        (* Output: *)
        (* judge = *)
        (* 1 *)
        (* 'NearZero:15' judge = norm(near) < 1e-6; *)
        se3mat_0[0] := V[0];
        se3mat_0[1] := V[1];
        se3mat_0[2] := V[2];
        e_theta := norm(x := se3mat_0);
        IF ABS(e_theta) < 1.0E-6 THEN 
            (* 'MatrixExp6:24' T = [eye(3), se3mat(1: 3, 4); 0, 0, 0, 1]; *)
            i0_eye();
            tmp_0 := i0_eye.I;
            FOR Slist_tmp_0 := 0 TO 2 DO 
                R_tmp := DWORD_TO_DINT(SHL(DINT_TO_DWORD(Slist_tmp_0), 2));
                a[R_tmp] := tmp_0[3 * Slist_tmp_0];
                a[R_tmp + 1] := tmp_0[(3 * Slist_tmp_0) + 1];
                a[R_tmp + 2] := tmp_0[(3 * Slist_tmp_0) + 2];
                a[Slist_tmp_0 + 12] := se3mat[Slist_tmp_0 + 12];
            END_FOR;
            a[3] := 0.0;
            a[7] := 0.0;
            a[11] := 0.0;
            a[15] := 1.0;
        ELSE 
            (* 'MatrixExp6:25' else *)
            (* 'MatrixExp6:26' [omghat, theta] = AxisAng3(omgtheta); *)
            (* *** CHAPTER 3: RIGID-BODY MOTIONS *** *)
            (* Takes A 3-vector of exponential coordinates for rotation. *)
            (* Returns the unit rotation axis omghat and the corresponding rotation  *)
            (* angle theta. *)
            (* Example Input: *)
            
            (* clear; clc; *)
            (* expc3 = [1; 2; 3]; *)
            (* [omghat, theta] = AxisAng3(expc3)   *)
            
            (* Output: *)
            (* omghat = *)
            (* 0.2673 *)
            (* 0.5345 *)
            (* 0.8018 *)
            (* theta = *)
            (* 3.7417 *)
            (* 'AxisAng3:20' theta = norm(expc3); *)
            (* 'AxisAng3:21' omghat = expc3 / theta; *)
            (* 'MatrixExp6:27' omgmat = se3mat(1: 3, 1: 3) / theta; *)
            FOR Slist_tmp_0 := 0 TO 2 DO 
                omgmat_tmp := DWORD_TO_DINT(SHL(DINT_TO_DWORD(Slist_tmp_0), 2));
                omgmat[3 * Slist_tmp_0] := se3mat[omgmat_tmp] / e_theta;
                omgmat[(3 * Slist_tmp_0) + 1] := se3mat[omgmat_tmp + 1] / e_theta;
                omgmat[(3 * Slist_tmp_0) + 2] := se3mat[omgmat_tmp + 2] / e_theta;
            END_FOR;
            (* 'MatrixExp6:28' T = [MatrixExp3(se3mat(1: 3, 1: 3)), ... *)
            (* 'MatrixExp6:29'          (eye(3) * theta + (1 - cos(theta)) * omgmat ... *)
            (* 'MatrixExp6:30'           + (theta - sin(theta)) * omgmat * omgmat) ... *)
            (* 'MatrixExp6:31'             * se3mat(1: 3, 4) / theta; *)
            (* 'MatrixExp6:32'          0, 0, 0, 1]; *)
            thetalist0_0 := 1.0 - COS(e_theta);
            g_a := e_theta - SIN(e_theta);
            (* *** CHAPTER 3: RIGID-BODY MOTIONS *** *)
            (* Takes a 3x3 so(3) representation of exponential coordinates. *)
            (* Returns R in SO(3) that is achieved by rotating about omghat by theta  *)
            (* from an initial orientation R = I. *)
            (* Example Input: *)
            
            (* clear; clc; *)
            (* so3mat = [[0, -3, 2]; [3, 0, -1]; [-2, 1, 0]]; *)
            (* R = MatrixExp3(so3mat)   *)
            
            (* Output: *)
            (* R = *)
            (* -0.6949    0.7135    0.0893 *)
            (* -0.1920   -0.3038    0.9332 *)
            (* 0.6930    0.6313    0.3481 *)
            (* 'MatrixExp3:18' omgtheta = so3ToVec(so3mat); *)
            (* *** CHAPTER 3: RIGID-BODY MOTIONS *** *)
            (* Takes a 3x3 skew-symmetric matrix (an element of so(3)). *)
            (* Returns the corresponding 3-vector (angular velocity). *)
            (* Example Input:  *)
            
            (* clear; clc; *)
            (* so3mat = [[0, -3, 2]; [3, 0, -1]; [-2, 1, 0]]; *)
            (* omg = so3ToVec(so3mat)   *)
            
            (* Output: *)
            (* omg = *)
            (* 1 *)
            (* 2 *)
            (* 3 *)
            (* 'so3ToVec:17' omg = [so3mat(3, 2); so3mat(1, 3); so3mat(2, 1)]; *)
            (* 'MatrixExp3:19' if NearZero(norm(omgtheta)) *)
            (* *** BASIC HELPER FUNCTIONS *** *)
            (* Takes a scalar. *)
            (* Checks if the scalar is small enough to be neglected. *)
            (* Example Input: *)
            
            (* clear; clc; *)
            (* near = -1e-7; *)
            (* judge = NearZero(near) *)
            
            (* Output: *)
            (* judge = *)
            (* 1 *)
            (* 'NearZero:15' judge = norm(near) < 1e-6; *)
            se3mat_0[0] := V[0];
            se3mat_0[1] := V[1];
            se3mat_0[2] := V[2];
            h_theta := norm(x := se3mat_0);
            IF ABS(h_theta) < 1.0E-6 THEN 
                (* 'MatrixExp3:20' R = eye(3); *)
                i0_eye();
                b_R := i0_eye.I;
            ELSE 
                (* 'MatrixExp3:21' else *)
                (* 'MatrixExp3:22' [omghat, theta] = AxisAng3(omgtheta); *)
                (* *** CHAPTER 3: RIGID-BODY MOTIONS *** *)
                (* Takes A 3-vector of exponential coordinates for rotation. *)
                (* Returns the unit rotation axis omghat and the corresponding rotation  *)
                (* angle theta. *)
                (* Example Input: *)
                
                (* clear; clc; *)
                (* expc3 = [1; 2; 3]; *)
                (* [omghat, theta] = AxisAng3(expc3)   *)
                
                (* Output: *)
                (* omghat = *)
                (* 0.2673 *)
                (* 0.5345 *)
                (* 0.8018 *)
                (* theta = *)
                (* 3.7417 *)
                (* 'AxisAng3:20' theta = norm(expc3); *)
                (* 'AxisAng3:21' omghat = expc3 / theta; *)
                (* 'MatrixExp3:23' omgmat = so3mat / theta; *)
                FOR Slist_tmp_0 := 0 TO 2 DO 
                    omgmat_tmp := DWORD_TO_DINT(SHL(DINT_TO_DWORD(Slist_tmp_0), 2));
                    b_omgmat[3 * Slist_tmp_0] := se3mat[omgmat_tmp] / h_theta;
                    b_omgmat[(3 * Slist_tmp_0) + 1] := se3mat[omgmat_tmp + 1] / h_theta;
                    b_omgmat[(3 * Slist_tmp_0) + 2] := se3mat[omgmat_tmp + 2] / h_theta;
                END_FOR;
                (* 'MatrixExp3:24' R = eye(3) + sin(theta) * omgmat + (1 - cos(theta)) * omgmat * omgmat; *)
                l_a := SIN(h_theta);
                x_tmp := COS(h_theta);
                i0_eye();
                tmp_0 := i0_eye.I;
                FOR Slist_tmp_0 := 0 TO 2 DO 
                    FOR omgmat_tmp := 0 TO 2 DO 
                        R_tmp := (3 * omgmat_tmp) + Slist_tmp_0;
                        b_R[R_tmp] := (((((1.0 - x_tmp) * b_omgmat[Slist_tmp_0 + 3]) * b_omgmat[(3 * omgmat_tmp) + 1]) + (((1.0 - x_tmp) * b_omgmat[Slist_tmp_0]) * b_omgmat[3 * omgmat_tmp])) + ((b_omgmat[Slist_tmp_0 + 6] * (1.0 - x_tmp)) * b_omgmat[(3 * omgmat_tmp) + 2])) + ((b_omgmat[R_tmp] * l_a) + tmp_0[R_tmp]);
                    END_FOR;
                END_FOR;
            END_IF;
            FOR Slist_tmp_0 := 0 TO 2 DO 
                l_a := 0.0;
                FOR omgmat_tmp := 0 TO 2 DO 
                    R_tmp := (3 * omgmat_tmp) + Slist_tmp_0;
                    l_a := ((((((omgmat[Slist_tmp_0 + 3] * g_a) * omgmat[(3 * omgmat_tmp) + 1]) + ((g_a * omgmat[Slist_tmp_0]) * omgmat[3 * omgmat_tmp])) + ((omgmat[Slist_tmp_0 + 6] * g_a) * omgmat[(3 * omgmat_tmp) + 2])) + ((SINT_TO_LREAL(p_a[R_tmp]) * e_theta) + (omgmat[R_tmp] * thetalist0_0))) * se3mat[omgmat_tmp + 12]) + l_a;
                    a[omgmat_tmp + (Slist_tmp_0 * 4)] := b_R[(3 * Slist_tmp_0) + omgmat_tmp];
                END_FOR;
                a[Slist_tmp_0 + 12] := l_a / e_theta;
            END_FOR;
            a[3] := 0.0;
            a[7] := 0.0;
            a[11] := 0.0;
            a[15] := 1.0;
        END_IF;
        FOR Slist_tmp_0 := 0 TO 3 DO 
            FOR omgmat_tmp := 0 TO 3 DO 
                a_tmp_tmp := DWORD_TO_DINT(SHL(DINT_TO_DWORD(omgmat_tmp), 2));
                R_tmp := Slist_tmp_0 + a_tmp_tmp;
                b_T[R_tmp] := 0.0;
                b_T[R_tmp] := b_T[R_tmp] + (a[a_tmp_tmp] * a_0[Slist_tmp_0]);
                b_T[R_tmp] := (a[a_tmp_tmp + 1] * a_0[Slist_tmp_0 + 4]) + b_T[R_tmp];
                b_T[R_tmp] := (a[a_tmp_tmp + 2] * a_0[Slist_tmp_0 + 8]) + b_T[R_tmp];
                b_T[R_tmp] := (a[a_tmp_tmp + 3] * a_0[Slist_tmp_0 + 12]) + b_T[R_tmp];
            END_FOR;
        END_FOR;
        FOR Slist_tmp_0 := 0 TO 15 DO 
            a_0[Slist_tmp_0] := b_T[Slist_tmp_0];
        END_FOR;
        (* 'JacobianSpace:31' Js(:, i) = Adjoint(T) * Slist(:, i); *)
        (* *** CHAPTER 3: RIGID-BODY MOTIONS *** *)
        (* Takes T a transformation matrix SE3.  *)
        (* Returns the corresponding 6x6 adjoint representation [AdT]. *)
        (* Example Input: *)
        
        (* clear; clc; *)
        (* T = [[1, 0, 0, 0]; [0, 0, -1, 0]; [0, 1, 0, 3]; [0, 0, 0, 1]]; *)
        (* AdT = Adjoint(T) *)
        
        (* Output: *)
        (* AdT = *)
        (* 1     0     0     0     0     0 *)
        (* 0     0    -1     0     0     0 *)
        (* 0     1     0     0     0     0 *)
        (* 0     0     3     1     0     0 *)
        (* 3     0     0     0     0    -1 *)
        (* 0     0     0     0     1     0 *)
        (* 'Adjoint:20' [R, p] = TransToRp(T); *)
        (* *** CHAPTER 3: RIGID-BODY MOTIONS *** *)
        (* Takes the transformation matrix T in SE(3)  *)
        (* Returns R: the corresponding rotation matrix *)
        (* p: the corresponding position vector . *)
        (* Example Input: *)
        
        (* clear; clc; *)
        (* T = [[1, 0, 0, 0]; [0, 0, -1, 0]; [0, 1, 0, 3]; [0, 0, 0, 1]]; *)
        (* [R, p] = TransToRp(T) *)
        
        (* Output: *)
        (* R = *)
        (* 1     0     0 *)
        (* 0     0    -1 *)
        (* 0     1     0 *)
        (* p = *)
        (* 0 *)
        (* 0 *)
        (* 3 *)
        (* 'TransToRp:22' R = T(1: 3, 1: 3); *)
        (* 'TransToRp:23' p = T(1: 3, 4); *)
        (* 'Adjoint:21' AdT = [R, zeros(3); VecToso3(p) * R, R]; *)
        (* *** CHAPTER 3: RIGID-BODY MOTIONS *** *)
        (* Takes a 3-vector (angular velocity). *)
        (* Returns the skew symmetric matrix in so(3). *)
        (* Example Input: *)
        
        (* clear; clc; *)
        (* omg = [1; 2; 3]; *)
        (* so3mat = VecToso3(omg) *)
        
        (* Output: *)
        (* so3mat = *)
        (* 0    -3     2 *)
        (* 3     0    -1 *)
        (* -2     1     0 *)
        (* 'VecToso3:17' so3mat = [0, -omg(3), omg(2); omg(3), 0, -omg(1); -omg(2), omg(1), 0]; *)
        tmp_3[3] :=  -a_0[14];
        tmp_3[6] := a_0[13];
        tmp_3[1] := a_0[14];
        tmp_3[7] :=  -a_0[12];
        tmp_3[2] :=  -a_0[13];
        tmp_3[5] := a_0[12];
        FOR Slist_tmp_0 := 0 TO 2 DO 
            FOR omgmat_tmp := 0 TO 2 DO 
                R_tmp := Slist_tmp_0 + (3 * omgmat_tmp);
                tmp_0[R_tmp] := 0.0;
                a_tmp_tmp := DWORD_TO_DINT(SHL(DINT_TO_DWORD(omgmat_tmp), 2));
                tmp_0[R_tmp] := tmp_0[R_tmp] + (a_0[a_tmp_tmp] * tmp_3[Slist_tmp_0]);
                tmp_0[R_tmp] := (a_0[a_tmp_tmp + 1] * tmp_3[Slist_tmp_0 + 3]) + tmp_0[R_tmp];
                tmp_0[R_tmp] := (a_0[a_tmp_tmp + 2] * tmp_3[Slist_tmp_0 + 6]) + tmp_0[R_tmp];
                Tsb_0[omgmat_tmp + (6 * Slist_tmp_0)] := a_0[(Slist_tmp_0 * 4) + omgmat_tmp];
                Tsb_0[omgmat_tmp + (6 * (Slist_tmp_0 + 3))] := 0.0;
            END_FOR;
        END_FOR;
        FOR Slist_tmp_0 := 0 TO 2 DO 
            Tsb_0[(6 * Slist_tmp_0) + 3] := tmp_0[3 * Slist_tmp_0];
            R_tmp := DWORD_TO_DINT(SHL(DINT_TO_DWORD(Slist_tmp_0), 2));
            omgmat_tmp := 6 * (Slist_tmp_0 + 3);
            Tsb_0[omgmat_tmp + 3] := a_0[R_tmp];
            Tsb_0[(6 * Slist_tmp_0) + 4] := tmp_0[(3 * Slist_tmp_0) + 1];
            Tsb_0[omgmat_tmp + 4] := a_0[R_tmp + 1];
            Tsb_0[(6 * Slist_tmp_0) + 5] := tmp_0[(3 * Slist_tmp_0) + 2];
            Tsb_0[omgmat_tmp + 5] := a_0[R_tmp + 2];
        END_FOR;
        FOR Slist_tmp_0 := 0 TO 5 DO 
            R_tmp := 6 * (d_i + 1);
            a_tmp_tmp := Slist_tmp_0 + R_tmp;
            Js[a_tmp_tmp] := 0.0;
            FOR omgmat_tmp := 0 TO 5 DO 
                Js[a_tmp_tmp] := (Slist[R_tmp + omgmat_tmp] * Tsb_0[(6 * omgmat_tmp) + Slist_tmp_0]) + Js[a_tmp_tmp];
            END_FOR;
        END_FOR;
    END_FOR;
    i0_pinv(A := Js);
    tmp_1 := i0_pinv.X;
    FOR Slist_tmp_0 := 0 TO 4 DO 
        l_a := 0.0;
        FOR omgmat_tmp := 0 TO 5 DO 
            l_a := (tmp_1[(5 * omgmat_tmp) + Slist_tmp_0] * Vs[omgmat_tmp]) + l_a;
        END_FOR;
        thetalist0[Slist_tmp_0] := thetalist0[Slist_tmp_0] + l_a;
    END_FOR;
    (* 'IKinSpace:57' thetalistDot = pinv(JacobianSpace(Slist, thetalist)) * Vs; *)
    (* *** CHAPTER 5: VELOCITY KINEMATICS AND STATICS *** *)
    (* Takes Slist: The joint screw axes in the space frame when the manipulator *)
    (* is at the home position, in the format of a matrix with the *)
    (* screw axes as the columns, *)
    (* thetalist: A list of joint coordinates.  *)
    (* Returns the corresponding space Jacobian (6xn real numbers). *)
    (* Example Input: *)
    
    (* clear; clc; *)
    (* Slist = [[0; 0; 1;   0; 0.2; 0.2], ... *)
    (* [1; 0; 0;   2;   0;   3], ... *)
    (* [0; 1; 0;   0;   2;   1], ... *)
    (* [1; 0; 0; 0.2; 0.3; 0.4]]; *)
    (* thetalist = [0.2; 1.1; 0.1; 1.2]; *)
    (* Js = JacobianSpace(Slist, thetalist) *)
    
    (* Output: *)
    (* Js = *)
    (* 0    0.9801   -0.0901    0.9575 *)
    (* 0    0.1987    0.4446    0.2849 *)
    (* 1.0000         0    0.8912   -0.0453 *)
    (* 0    1.9522   -2.2164   -0.5116 *)
    (* 0.2000    0.4365   -2.4371    2.7754 *)
    (* 0.2000    2.9603    3.2357    2.2251 *)
    (* 'JacobianSpace:27' Js = Slist; *)
    (* 'JacobianSpace:28' T = eye(4); *)
    (* 'JacobianSpace:29' for i = 2: length(thetalist) *)
    (* 'IKinSpace:58' i = i + 1; *)
    i := i + 1;
    (* 'IKinSpace:59' Tsb = FKinSpace(M, Slist, thetalist); *)
    FOR Slist_tmp_0 := 0 TO 15 DO 
        Tsb[Slist_tmp_0] := M[Slist_tmp_0];
    END_FOR;
    (* *** CHAPTER 4: FORWARD KINEMATICS *** *)
    (* Takes M: the home configuration (position and orientation) of the  *)
    (* end-effector, *)
    (* Slist: The joint screw axes in the space frame when the manipulator *)
    (* is at the home position, *)
    (* thetalist: A list of joint coordinates. *)
    (* Returns T in SE(3) representing the end-effector frame, when the joints  *)
    (* are at the specified coordinates (i.t.o Space Frame). *)
    (* Example Inputs: *)
    
    (* clear; clc; *)
    (* M = [[-1, 0, 0, 0]; [0, 1, 0, 6]; [0, 0, -1, 2]; [0, 0, 0, 1]]; *)
    (* Slist = [[0; 0;  1;  4; 0;    0], ... *)
    (* [0; 0;  0;  0; 1;    0], ... *)
    (* [0; 0; -1; -6; 0; -0.1]]; *)
    (* thetalist =[pi / 2; 3; pi]; *)
    (* T = FKinSpace(M, Slist, thetalist) *)
    
    (* Output: *)
    (* T = *)
    (* -0.0000    1.0000         0   -5.0000 *)
    (* 1.0000    0.0000         0    4.0000 *)
    (* 0         0   -1.0000    1.6858 *)
    (* 0         0         0    1.0000 *)
    (* 'FKinSpace:27' T = M; *)
    (* 'FKinSpace:28' for i = size(thetalist,1): -1: 1 *)
    se3mat[0] := 0.0;
    se3mat[5] := 0.0;
    se3mat[10] := 0.0;
    se3mat[3] := 0.0;
    se3mat[7] := 0.0;
    se3mat[11] := 0.0;
    se3mat[15] := 0.0;
    FOR e_i := 0 TO 4 DO 
        (* 'FKinSpace:29' T = MatrixExp6(VecTose3(Slist(:, i) * thetalist(i))) * T; *)
        thetalist0_0 := thetalist0[4 - e_i];
        FOR Slist_tmp_0 := 0 TO 5 DO 
            V[Slist_tmp_0] := Slist[((4 - e_i) * 6) + Slist_tmp_0] * thetalist0_0;
        END_FOR;
        (* *** CHAPTER 3: RIGID-BODY MOTIONS *** *)
        (* Takes a 6-vector (representing a spatial velocity). *)
        (* Returns the corresponding 4x4 se(3) matrix. *)
        (* Example Input: *)
        
        (* clear; clc; *)
        (* V = [1; 2; 3; 4; 5; 6]; *)
        (* se3mat = VecTose3(V) *)
        
        (* Output: *)
        (* se3mat = *)
        (* 0    -3     2     4 *)
        (* 3     0    -1     5 *)
        (* -2     1     0     6 *)
        (* 0     0     0     0  *)
        (* 'VecTose3:18' se3mat = [VecToso3(V(1: 3)), V(4: 6); 0, 0, 0, 0]; *)
        (* *** CHAPTER 3: RIGID-BODY MOTIONS *** *)
        (* Takes a 3-vector (angular velocity). *)
        (* Returns the skew symmetric matrix in so(3). *)
        (* Example Input: *)
        
        (* clear; clc; *)
        (* omg = [1; 2; 3]; *)
        (* so3mat = VecToso3(omg) *)
        
        (* Output: *)
        (* so3mat = *)
        (* 0    -3     2 *)
        (* 3     0    -1 *)
        (* -2     1     0 *)
        (* 'VecToso3:17' so3mat = [0, -omg(3), omg(2); omg(3), 0, -omg(1); -omg(2), omg(1), 0]; *)
        se3mat[4] :=  -V[2];
        se3mat[8] := V[1];
        se3mat[1] := V[2];
        se3mat[9] :=  -V[0];
        se3mat[2] :=  -V[1];
        se3mat[6] := V[0];
        se3mat[12] := V[3];
        se3mat[13] := V[4];
        se3mat[14] := V[5];
        (* *** CHAPTER 3: RIGID-BODY MOTIONS *** *)
        (* Takes a se(3) representation of exponential coordinates. *)
        (* Returns a T matrix in SE(3) that is achieved by traveling along/about the  *)
        (* screw axis S for a distance theta from an initial configuration T = I. *)
        (* Example Input: *)
        
        (* clear; clc; *)
        (* se3mat = [ 0,      0,       0,      0; *)
        (* 0,      0, -1.5708, 2.3562; *)
        (* 0, 1.5708,       0, 2.3562; *)
        (* 0,      0,       0,      0] *)
        (* T = MatrixExp6(se3mat) *)
        
        (* Output: *)
        (* T = *)
        (* 1.0000         0         0         0 *)
        (* 0    0.0000   -1.0000   -0.0000 *)
        (* 0    1.0000    0.0000    3.0000 *)
        (* 0         0         0    1.0000  *)
        (* 'MatrixExp6:22' omgtheta = so3ToVec(se3mat(1: 3, 1: 3)); *)
        (* *** CHAPTER 3: RIGID-BODY MOTIONS *** *)
        (* Takes a 3x3 skew-symmetric matrix (an element of so(3)). *)
        (* Returns the corresponding 3-vector (angular velocity). *)
        (* Example Input:  *)
        
        (* clear; clc; *)
        (* so3mat = [[0, -3, 2]; [3, 0, -1]; [-2, 1, 0]]; *)
        (* omg = so3ToVec(so3mat)   *)
        
        (* Output: *)
        (* omg = *)
        (* 1 *)
        (* 2 *)
        (* 3 *)
        (* 'so3ToVec:17' omg = [so3mat(3, 2); so3mat(1, 3); so3mat(2, 1)]; *)
        omgtheta[0] := V[0];
        omgtheta[1] := V[1];
        omgtheta[2] := V[2];
        (* 'MatrixExp6:23' if NearZero(norm(omgtheta)) *)
        (* *** BASIC HELPER FUNCTIONS *** *)
        (* Takes a scalar. *)
        (* Checks if the scalar is small enough to be neglected. *)
        (* Example Input: *)
        
        (* clear; clc; *)
        (* near = -1e-7; *)
        (* judge = NearZero(near) *)
        
        (* Output: *)
        (* judge = *)
        (* 1 *)
        (* 'NearZero:15' judge = norm(near) < 1e-6; *)
        f_theta := norm(x := omgtheta);
        IF ABS(f_theta) < 1.0E-6 THEN 
            (* 'MatrixExp6:24' T = [eye(3), se3mat(1: 3, 4); 0, 0, 0, 1]; *)
            i0_eye();
            tmp_0 := i0_eye.I;
            FOR Slist_tmp_0 := 0 TO 2 DO 
                R_tmp := DWORD_TO_DINT(SHL(DINT_TO_DWORD(Slist_tmp_0), 2));
                a[R_tmp] := tmp_0[3 * Slist_tmp_0];
                a[R_tmp + 1] := tmp_0[(3 * Slist_tmp_0) + 1];
                a[R_tmp + 2] := tmp_0[(3 * Slist_tmp_0) + 2];
                a[Slist_tmp_0 + 12] := se3mat[Slist_tmp_0 + 12];
            END_FOR;
            a[3] := 0.0;
            a[7] := 0.0;
            a[11] := 0.0;
            a[15] := 1.0;
        ELSE 
            (* 'MatrixExp6:25' else *)
            (* 'MatrixExp6:26' [omghat, theta] = AxisAng3(omgtheta); *)
            (* *** CHAPTER 3: RIGID-BODY MOTIONS *** *)
            (* Takes A 3-vector of exponential coordinates for rotation. *)
            (* Returns the unit rotation axis omghat and the corresponding rotation  *)
            (* angle theta. *)
            (* Example Input: *)
            
            (* clear; clc; *)
            (* expc3 = [1; 2; 3]; *)
            (* [omghat, theta] = AxisAng3(expc3)   *)
            
            (* Output: *)
            (* omghat = *)
            (* 0.2673 *)
            (* 0.5345 *)
            (* 0.8018 *)
            (* theta = *)
            (* 3.7417 *)
            (* 'AxisAng3:20' theta = norm(expc3); *)
            (* 'AxisAng3:21' omghat = expc3 / theta; *)
            (* 'MatrixExp6:27' omgmat = se3mat(1: 3, 1: 3) / theta; *)
            FOR Slist_tmp_0 := 0 TO 2 DO 
                omgmat_tmp := DWORD_TO_DINT(SHL(DINT_TO_DWORD(Slist_tmp_0), 2));
                omgmat[3 * Slist_tmp_0] := se3mat[omgmat_tmp] / f_theta;
                omgmat[(3 * Slist_tmp_0) + 1] := se3mat[omgmat_tmp + 1] / f_theta;
                omgmat[(3 * Slist_tmp_0) + 2] := se3mat[omgmat_tmp + 2] / f_theta;
            END_FOR;
            (* 'MatrixExp6:28' T = [MatrixExp3(se3mat(1: 3, 1: 3)), ... *)
            (* 'MatrixExp6:29'          (eye(3) * theta + (1 - cos(theta)) * omgmat ... *)
            (* 'MatrixExp6:30'           + (theta - sin(theta)) * omgmat * omgmat) ... *)
            (* 'MatrixExp6:31'             * se3mat(1: 3, 4) / theta; *)
            (* 'MatrixExp6:32'          0, 0, 0, 1]; *)
            thetalist0_0 := 1.0 - COS(f_theta);
            g_a := f_theta - SIN(f_theta);
            (* *** CHAPTER 3: RIGID-BODY MOTIONS *** *)
            (* Takes a 3x3 so(3) representation of exponential coordinates. *)
            (* Returns R in SO(3) that is achieved by rotating about omghat by theta  *)
            (* from an initial orientation R = I. *)
            (* Example Input: *)
            
            (* clear; clc; *)
            (* so3mat = [[0, -3, 2]; [3, 0, -1]; [-2, 1, 0]]; *)
            (* R = MatrixExp3(so3mat)   *)
            
            (* Output: *)
            (* R = *)
            (* -0.6949    0.7135    0.0893 *)
            (* -0.1920   -0.3038    0.9332 *)
            (* 0.6930    0.6313    0.3481 *)
            (* 'MatrixExp3:18' omgtheta = so3ToVec(so3mat); *)
            (* *** CHAPTER 3: RIGID-BODY MOTIONS *** *)
            (* Takes a 3x3 skew-symmetric matrix (an element of so(3)). *)
            (* Returns the corresponding 3-vector (angular velocity). *)
            (* Example Input:  *)
            
            (* clear; clc; *)
            (* so3mat = [[0, -3, 2]; [3, 0, -1]; [-2, 1, 0]]; *)
            (* omg = so3ToVec(so3mat)   *)
            
            (* Output: *)
            (* omg = *)
            (* 1 *)
            (* 2 *)
            (* 3 *)
            (* 'so3ToVec:17' omg = [so3mat(3, 2); so3mat(1, 3); so3mat(2, 1)]; *)
            (* 'MatrixExp3:19' if NearZero(norm(omgtheta)) *)
            (* *** BASIC HELPER FUNCTIONS *** *)
            (* Takes a scalar. *)
            (* Checks if the scalar is small enough to be neglected. *)
            (* Example Input: *)
            
            (* clear; clc; *)
            (* near = -1e-7; *)
            (* judge = NearZero(near) *)
            
            (* Output: *)
            (* judge = *)
            (* 1 *)
            (* 'NearZero:15' judge = norm(near) < 1e-6; *)
            se3mat_0[0] := V[0];
            se3mat_0[1] := V[1];
            se3mat_0[2] := V[2];
            j_theta := norm(x := se3mat_0);
            IF ABS(j_theta) < 1.0E-6 THEN 
                (* 'MatrixExp3:20' R = eye(3); *)
                i0_eye();
                b_R := i0_eye.I;
            ELSE 
                (* 'MatrixExp3:21' else *)
                (* 'MatrixExp3:22' [omghat, theta] = AxisAng3(omgtheta); *)
                (* *** CHAPTER 3: RIGID-BODY MOTIONS *** *)
                (* Takes A 3-vector of exponential coordinates for rotation. *)
                (* Returns the unit rotation axis omghat and the corresponding rotation  *)
                (* angle theta. *)
                (* Example Input: *)
                
                (* clear; clc; *)
                (* expc3 = [1; 2; 3]; *)
                (* [omghat, theta] = AxisAng3(expc3)   *)
                
                (* Output: *)
                (* omghat = *)
                (* 0.2673 *)
                (* 0.5345 *)
                (* 0.8018 *)
                (* theta = *)
                (* 3.7417 *)
                (* 'AxisAng3:20' theta = norm(expc3); *)
                (* 'AxisAng3:21' omghat = expc3 / theta; *)
                (* 'MatrixExp3:23' omgmat = so3mat / theta; *)
                FOR Slist_tmp_0 := 0 TO 2 DO 
                    omgmat_tmp := DWORD_TO_DINT(SHL(DINT_TO_DWORD(Slist_tmp_0), 2));
                    b_omgmat[3 * Slist_tmp_0] := se3mat[omgmat_tmp] / j_theta;
                    b_omgmat[(3 * Slist_tmp_0) + 1] := se3mat[omgmat_tmp + 1] / j_theta;
                    b_omgmat[(3 * Slist_tmp_0) + 2] := se3mat[omgmat_tmp + 2] / j_theta;
                END_FOR;
                (* 'MatrixExp3:24' R = eye(3) + sin(theta) * omgmat + (1 - cos(theta)) * omgmat * omgmat; *)
                l_a := SIN(j_theta);
                x_tmp := COS(j_theta);
                i0_eye();
                tmp_0 := i0_eye.I;
                FOR Slist_tmp_0 := 0 TO 2 DO 
                    FOR omgmat_tmp := 0 TO 2 DO 
                        R_tmp := (3 * omgmat_tmp) + Slist_tmp_0;
                        b_R[R_tmp] := (((((1.0 - x_tmp) * b_omgmat[Slist_tmp_0 + 3]) * b_omgmat[(3 * omgmat_tmp) + 1]) + (((1.0 - x_tmp) * b_omgmat[Slist_tmp_0]) * b_omgmat[3 * omgmat_tmp])) + ((b_omgmat[Slist_tmp_0 + 6] * (1.0 - x_tmp)) * b_omgmat[(3 * omgmat_tmp) + 2])) + ((b_omgmat[R_tmp] * l_a) + tmp_0[R_tmp]);
                    END_FOR;
                END_FOR;
            END_IF;
            FOR Slist_tmp_0 := 0 TO 2 DO 
                l_a := 0.0;
                FOR omgmat_tmp := 0 TO 2 DO 
                    R_tmp := (3 * omgmat_tmp) + Slist_tmp_0;
                    l_a := ((((((omgmat[Slist_tmp_0 + 3] * g_a) * omgmat[(3 * omgmat_tmp) + 1]) + ((g_a * omgmat[Slist_tmp_0]) * omgmat[3 * omgmat_tmp])) + ((omgmat[Slist_tmp_0 + 6] * g_a) * omgmat[(3 * omgmat_tmp) + 2])) + ((SINT_TO_LREAL(p_a[R_tmp]) * f_theta) + (omgmat[R_tmp] * thetalist0_0))) * se3mat[omgmat_tmp + 12]) + l_a;
                    a[omgmat_tmp + (Slist_tmp_0 * 4)] := b_R[(3 * Slist_tmp_0) + omgmat_tmp];
                END_FOR;
                a[Slist_tmp_0 + 12] := l_a / f_theta;
            END_FOR;
            a[3] := 0.0;
            a[7] := 0.0;
            a[11] := 0.0;
            a[15] := 1.0;
        END_IF;
        FOR Slist_tmp_0 := 0 TO 3 DO 
            FOR omgmat_tmp := 0 TO 3 DO 
                a_tmp_tmp := DWORD_TO_DINT(SHL(DINT_TO_DWORD(omgmat_tmp), 2));
                R_tmp := Slist_tmp_0 + a_tmp_tmp;
                a_0[R_tmp] := 0.0;
                a_0[R_tmp] := a_0[R_tmp] + (Tsb[a_tmp_tmp] * a[Slist_tmp_0]);
                a_0[R_tmp] := (Tsb[a_tmp_tmp + 1] * a[Slist_tmp_0 + 4]) + a_0[R_tmp];
                a_0[R_tmp] := (Tsb[a_tmp_tmp + 2] * a[Slist_tmp_0 + 8]) + a_0[R_tmp];
                a_0[R_tmp] := (Tsb[a_tmp_tmp + 3] * a[Slist_tmp_0 + 12]) + a_0[R_tmp];
            END_FOR;
        END_FOR;
        FOR Slist_tmp_0 := 0 TO 15 DO 
            Tsb[Slist_tmp_0] := a_0[Slist_tmp_0];
        END_FOR;
    END_FOR;
    (* 'IKinSpace:60' Vs = Adjoint(Tsb) * se3ToVec(MatrixLog6(TransInv(Tsb) * T)); *)
    (* *** CHAPTER 3: RIGID-BODY MOTIONS *** *)
    (* Takes a transformation matrix T. *)
    (* Returns its inverse.  *)
    (* Uses the structure of transformation matrices to avoid taking a matrix *)
    (* inverse, for efficiency. *)
    (* Example Input: *)
    
    (* clear; clc; *)
    (* T = [[1, 0, 0, 0]; [0, 0, -1, 0]; [0, 1, 0, 3]; [0, 0, 0, 1]]; *)
    (* invT = TransInv(T) *)
    
    (* Ouput: *)
    (* invT = *)
    (* 1     0     0     0 *)
    (* 0     0     1    -3 *)
    (* 0    -1     0     0 *)
    (* 0     0     0     1 *)
    (* 'TransInv:20' [R, p] = TransToRp(T); *)
    (* *** CHAPTER 3: RIGID-BODY MOTIONS *** *)
    (* Takes the transformation matrix T in SE(3)  *)
    (* Returns R: the corresponding rotation matrix *)
    (* p: the corresponding position vector . *)
    (* Example Input: *)
    
    (* clear; clc; *)
    (* T = [[1, 0, 0, 0]; [0, 0, -1, 0]; [0, 1, 0, 3]; [0, 0, 0, 1]]; *)
    (* [R, p] = TransToRp(T) *)
    
    (* Output: *)
    (* R = *)
    (* 1     0     0 *)
    (* 0     0    -1 *)
    (* 0     1     0 *)
    (* p = *)
    (* 0 *)
    (* 0 *)
    (* 3 *)
    (* 'TransToRp:22' R = T(1: 3, 1: 3); *)
    (* 'TransToRp:23' p = T(1: 3, 4); *)
    (* 'TransInv:21' invT = [transpose(R), -transpose(R) * p; 0, 0, 0, 1]; *)
    FOR Slist_tmp_0 := 0 TO 2 DO 
        omgmat[3 * Slist_tmp_0] := Tsb[Slist_tmp_0];
        omgmat[(3 * Slist_tmp_0) + 1] := Tsb[Slist_tmp_0 + 4];
        omgmat[(3 * Slist_tmp_0) + 2] := Tsb[Slist_tmp_0 + 8];
    END_FOR;
    FOR Slist_tmp_0 := 0 TO 8 DO 
        b_R[Slist_tmp_0] :=  -omgmat[Slist_tmp_0];
    END_FOR;
    FOR Slist_tmp_0 := 0 TO 2 DO 
        omgmat_tmp := DWORD_TO_DINT(SHL(DINT_TO_DWORD(Slist_tmp_0), 2));
        se3mat[omgmat_tmp] := omgmat[3 * Slist_tmp_0];
        se3mat[omgmat_tmp + 1] := omgmat[(3 * Slist_tmp_0) + 1];
        se3mat[omgmat_tmp + 2] := omgmat[(3 * Slist_tmp_0) + 2];
        se3mat[Slist_tmp_0 + 12] := (b_R[Slist_tmp_0 + 6] * Tsb[14]) + ((b_R[Slist_tmp_0 + 3] * Tsb[13]) + (b_R[Slist_tmp_0] * Tsb[12]));
    END_FOR;
    se3mat[3] := 0.0;
    se3mat[7] := 0.0;
    se3mat[11] := 0.0;
    se3mat[15] := 1.0;
    FOR Slist_tmp_0 := 0 TO 3 DO 
        FOR omgmat_tmp := 0 TO 3 DO 
            a_tmp_tmp := DWORD_TO_DINT(SHL(DINT_TO_DWORD(omgmat_tmp), 2));
            R_tmp := Slist_tmp_0 + a_tmp_tmp;
            a_0[R_tmp] := 0.0;
            a_0[R_tmp] := a_0[R_tmp] + (T[a_tmp_tmp] * se3mat[Slist_tmp_0]);
            a_0[R_tmp] := (T[a_tmp_tmp + 1] * se3mat[Slist_tmp_0 + 4]) + a_0[R_tmp];
            a_0[R_tmp] := (T[a_tmp_tmp + 2] * se3mat[Slist_tmp_0 + 8]) + a_0[R_tmp];
            a_0[R_tmp] := (T[a_tmp_tmp + 3] * se3mat[Slist_tmp_0 + 12]) + a_0[R_tmp];
        END_FOR;
    END_FOR;
    (* *** CHAPTER 3: RIGID-BODY MOTIONS *** *)
    (* Takes a transformation matrix T in SE(3). *)
    (* Returns the corresponding se(3) representation of exponential  *)
    (* coordinates. *)
    (* Example Input: *)
    
    (* clear; clc; *)
    (* T = [[1, 0, 0, 0]; [0, 0, -1, 0]; [0, 1, 0, 3]; [0, 0, 0, 1]]; *)
    (* expmat = MatrixLog6(T) *)
    
    (* Output: *)
    (* expc6 = *)
    (* 0         0         0         0 *)
    (* 0         0   -1.5708    2.3562 *)
    (* 0    1.5708         0    2.3562 *)
    (* 0         0         0         0 *)
    (* 'MatrixLog6:19' [R, p] = TransToRp(T); *)
    (* *** CHAPTER 3: RIGID-BODY MOTIONS *** *)
    (* Takes the transformation matrix T in SE(3)  *)
    (* Returns R: the corresponding rotation matrix *)
    (* p: the corresponding position vector . *)
    (* Example Input: *)
    
    (* clear; clc; *)
    (* T = [[1, 0, 0, 0]; [0, 0, -1, 0]; [0, 1, 0, 3]; [0, 0, 0, 1]]; *)
    (* [R, p] = TransToRp(T) *)
    
    (* Output: *)
    (* R = *)
    (* 1     0     0 *)
    (* 0     0    -1 *)
    (* 0     1     0 *)
    (* p = *)
    (* 0 *)
    (* 0 *)
    (* 3 *)
    (* 'TransToRp:22' R = T(1: 3, 1: 3); *)
    (* 'TransToRp:23' p = T(1: 3, 4); *)
    (* 'MatrixLog6:20' omgmat = MatrixLog3(R); *)
    FOR Slist_tmp_0 := 0 TO 2 DO 
        R_tmp := DWORD_TO_DINT(SHL(DINT_TO_DWORD(Slist_tmp_0), 2));
        b_R[3 * Slist_tmp_0] := a_0[R_tmp];
        b_R[(3 * Slist_tmp_0) + 1] := a_0[R_tmp + 1];
        b_R[(3 * Slist_tmp_0) + 2] := a_0[R_tmp + 2];
    END_FOR;
    i0_MatrixLog3(b_R := b_R);
    omgmat := i0_MatrixLog3.so3mat;
    (* 'MatrixLog6:21' if isequal(omgmat, zeros(3)) *)
    IF isequal(varargin_1 := omgmat, varargin_2 := tmp_4) THEN 
        (* 'MatrixLog6:22' expmat = [zeros(3), T(1: 3, 4); 0, 0, 0, 0]; *)
        FOR Slist_tmp_0 := 0 TO 2 DO 
            omgmat_tmp := DWORD_TO_DINT(SHL(DINT_TO_DWORD(Slist_tmp_0), 2));
            se3mat[omgmat_tmp] := 0.0;
            se3mat[omgmat_tmp + 1] := 0.0;
            se3mat[omgmat_tmp + 2] := 0.0;
            se3mat[Slist_tmp_0 + 12] := a_0[Slist_tmp_0 + 12];
        END_FOR;
        se3mat[3] := 0.0;
        se3mat[7] := 0.0;
        se3mat[11] := 0.0;
        se3mat[15] := 0.0;
    ELSE 
        (* 'MatrixLog6:23' else *)
        (* 'MatrixLog6:24' theta = acos((trace(R) - 1) / 2); *)
        b_theta := ACOS((((a_0[0] + a_0[5]) + a_0[10]) - 1.0) / 2.0);
        (* 'MatrixLog6:25' expmat = [omgmat, (eye(3) - omgmat / 2 ... *)
        (* 'MatrixLog6:26'                       + (1 / theta - cot(theta / 2) / 2) ... *)
        (* 'MatrixLog6:27'                         * omgmat * omgmat / theta) * p; *)
        (* 'MatrixLog6:28'               0, 0, 0, 0]; *)
        thetalist0_0 := (1.0 / b_theta) - ((1.0 / TAN(b_theta / 2.0)) / 2.0);
        i0_eye();
        tmp_0 := i0_eye.I;
        FOR Slist_tmp_0 := 0 TO 2 DO 
            se3mat_0[Slist_tmp_0] := 0.0;
            FOR omgmat_tmp := 0 TO 2 DO 
                se3mat[omgmat_tmp + (Slist_tmp_0 * 4)] := omgmat[(3 * Slist_tmp_0) + omgmat_tmp];
                R_tmp := (3 * omgmat_tmp) + Slist_tmp_0;
                se3mat_0[Slist_tmp_0] := (((((((omgmat[Slist_tmp_0 + 3] * thetalist0_0) * omgmat[(3 * omgmat_tmp) + 1]) + ((thetalist0_0 * omgmat[Slist_tmp_0]) * omgmat[3 * omgmat_tmp])) + ((omgmat[Slist_tmp_0 + 6] * thetalist0_0) * omgmat[(3 * omgmat_tmp) + 2])) / b_theta) + (tmp_0[R_tmp] - (omgmat[R_tmp] / 2.0))) * a_0[omgmat_tmp + 12]) + se3mat_0[Slist_tmp_0];
            END_FOR;
            se3mat[Slist_tmp_0 + 12] := se3mat_0[Slist_tmp_0];
        END_FOR;
        se3mat[3] := 0.0;
        se3mat[7] := 0.0;
        se3mat[11] := 0.0;
        se3mat[15] := 0.0;
    END_IF;
    (* *** CHAPTER 3: RIGID-BODY MOTIONS *** *)
    (* Takes T a transformation matrix SE3.  *)
    (* Returns the corresponding 6x6 adjoint representation [AdT]. *)
    (* Example Input: *)
    
    (* clear; clc; *)
    (* T = [[1, 0, 0, 0]; [0, 0, -1, 0]; [0, 1, 0, 3]; [0, 0, 0, 1]]; *)
    (* AdT = Adjoint(T) *)
    
    (* Output: *)
    (* AdT = *)
    (* 1     0     0     0     0     0 *)
    (* 0     0    -1     0     0     0 *)
    (* 0     1     0     0     0     0 *)
    (* 0     0     3     1     0     0 *)
    (* 3     0     0     0     0    -1 *)
    (* 0     0     0     0     1     0 *)
    (* 'Adjoint:20' [R, p] = TransToRp(T); *)
    (* *** CHAPTER 3: RIGID-BODY MOTIONS *** *)
    (* Takes the transformation matrix T in SE(3)  *)
    (* Returns R: the corresponding rotation matrix *)
    (* p: the corresponding position vector . *)
    (* Example Input: *)
    
    (* clear; clc; *)
    (* T = [[1, 0, 0, 0]; [0, 0, -1, 0]; [0, 1, 0, 3]; [0, 0, 0, 1]]; *)
    (* [R, p] = TransToRp(T) *)
    
    (* Output: *)
    (* R = *)
    (* 1     0     0 *)
    (* 0     0    -1 *)
    (* 0     1     0 *)
    (* p = *)
    (* 0 *)
    (* 0 *)
    (* 3 *)
    (* 'TransToRp:22' R = T(1: 3, 1: 3); *)
    (* 'TransToRp:23' p = T(1: 3, 4); *)
    (* 'Adjoint:21' AdT = [R, zeros(3); VecToso3(p) * R, R]; *)
    (* *** CHAPTER 3: RIGID-BODY MOTIONS *** *)
    (* Takes a 3-vector (angular velocity). *)
    (* Returns the skew symmetric matrix in so(3). *)
    (* Example Input: *)
    
    (* clear; clc; *)
    (* omg = [1; 2; 3]; *)
    (* so3mat = VecToso3(omg) *)
    
    (* Output: *)
    (* so3mat = *)
    (* 0    -3     2 *)
    (* 3     0    -1 *)
    (* -2     1     0 *)
    (* 'VecToso3:17' so3mat = [0, -omg(3), omg(2); omg(3), 0, -omg(1); -omg(2), omg(1), 0]; *)
    (* *** CHAPTER 3: RIGID-BODY MOTIONS *** *)
    (* Takes se3mat a 4x4 se(3) matrix *)
    (* Returns the corresponding 6-vector (representing spatial velocity). *)
    (* Example Input: *)
    
    (* clear; clc; *)
    (* se3mat = [[0, -3, 2, 4]; [3, 0, -1, 5]; [-2, 1, 0, 6]; [0, 0, 0, 0]]; *)
    (* V = se3ToVec(se3mat) *)
    
    (* Output: *)
    (* V = *)
    (* 1 *)
    (* 2 *)
    (* 3 *)
    (* 4 *)
    (* 5 *)
    (* 6 *)
    (* 'se3ToVec:20' V = [se3mat(3, 2); se3mat(1, 3); se3mat(2, 1); se3mat(1: 3, 4)]; *)
    tmp_5[3] :=  -Tsb[14];
    tmp_5[6] := Tsb[13];
    tmp_5[1] := Tsb[14];
    tmp_5[7] :=  -Tsb[12];
    tmp_5[2] :=  -Tsb[13];
    tmp_5[5] := Tsb[12];
    FOR Slist_tmp_0 := 0 TO 2 DO 
        FOR omgmat_tmp := 0 TO 2 DO 
            R_tmp := Slist_tmp_0 + (3 * omgmat_tmp);
            tmp_0[R_tmp] := 0.0;
            a_tmp_tmp := DWORD_TO_DINT(SHL(DINT_TO_DWORD(omgmat_tmp), 2));
            tmp_0[R_tmp] := tmp_0[R_tmp] + (Tsb[a_tmp_tmp] * tmp_5[Slist_tmp_0]);
            tmp_0[R_tmp] := (Tsb[a_tmp_tmp + 1] * tmp_5[Slist_tmp_0 + 3]) + tmp_0[R_tmp];
            tmp_0[R_tmp] := (Tsb[a_tmp_tmp + 2] * tmp_5[Slist_tmp_0 + 6]) + tmp_0[R_tmp];
            Tsb_0[omgmat_tmp + (6 * Slist_tmp_0)] := Tsb[(Slist_tmp_0 * 4) + omgmat_tmp];
            Tsb_0[omgmat_tmp + (6 * (Slist_tmp_0 + 3))] := 0.0;
        END_FOR;
    END_FOR;
    V[0] := se3mat[6];
    V[1] := se3mat[8];
    V[2] := se3mat[1];
    FOR Slist_tmp_0 := 0 TO 2 DO 
        Tsb_0[(6 * Slist_tmp_0) + 3] := tmp_0[3 * Slist_tmp_0];
        omgmat_tmp := DWORD_TO_DINT(SHL(DINT_TO_DWORD(Slist_tmp_0), 2));
        R_tmp := 6 * (Slist_tmp_0 + 3);
        Tsb_0[R_tmp + 3] := Tsb[omgmat_tmp];
        Tsb_0[(6 * Slist_tmp_0) + 4] := tmp_0[(3 * Slist_tmp_0) + 1];
        Tsb_0[R_tmp + 4] := Tsb[omgmat_tmp + 1];
        Tsb_0[(6 * Slist_tmp_0) + 5] := tmp_0[(3 * Slist_tmp_0) + 2];
        Tsb_0[R_tmp + 5] := Tsb[omgmat_tmp + 2];
        V[Slist_tmp_0 + 3] := se3mat[Slist_tmp_0 + 12];
    END_FOR;
    FOR Slist_tmp_0 := 0 TO 5 DO 
        Vs[Slist_tmp_0] := 0.0;
        FOR omgmat_tmp := 0 TO 5 DO 
            Vs[Slist_tmp_0] := (Tsb_0[(6 * omgmat_tmp) + Slist_tmp_0] * V[omgmat_tmp]) + Vs[Slist_tmp_0];
        END_FOR;
    END_FOR;
    (* 'IKinSpace:61' err = norm(Vs(1: 3)) > eomg || norm(Vs(4: 6)) > ev; *)
    se3mat_0[0] := Vs[0];
    se3mat_0[1] := Vs[1];
    se3mat_0[2] := Vs[2];
    IF norm(x := se3mat_0) <= 1.0E-5 THEN 
        se3mat_0[0] := Vs[3];
        se3mat_0[1] := Vs[4];
        se3mat_0[2] := Vs[5];
        IF norm(x := se3mat_0) <= 1.0E-7 THEN 
            err := FALSE;
        END_IF;
    END_IF;
END_WHILE;
(* 'IKinSpace:63' success = ~ err; *)
(* For velocity Kinematics 4 dof. *)
(* '<S1>:1:70' Vs = [0; 0;0; Vx; Vy; Vz]; *)
(* '<S1>:1:71' thetalist0_4DOF = [q1Inn; q2Inn; q3Inn; q4Inn; q5Inn; q6Inn]; *)
Vs[0] := q1Inn;
Vs[1] := q2Inn;
Vs[2] := q3Inn;
Vs[3] := q4Inn;
Vs[4] := q5Inn;
Vs[5] :=  -q1Inn;
(* '<S1>:1:72' Slist_4DOF = [S1,S2,S3,S4,S5,S6]; *)
(* MATLAB Function: '<Root>/MATLAB Function3' *)
FOR Slist_tmp_0 := 0 TO 5 DO 
    Tsb_0[Slist_tmp_0] := SINT_TO_LREAL(Slist_tmp[Slist_tmp_0]);
    Tsb_0[Slist_tmp_0 + 6] := g[Slist_tmp_0];
    Tsb_0[Slist_tmp_0 + 12] := h[Slist_tmp_0];
    Tsb_0[Slist_tmp_0 + 18] := SINT_TO_LREAL(b_l[Slist_tmp_0]);
    Tsb_0[Slist_tmp_0 + 24] := S5[Slist_tmp_0];
    Tsb_0[Slist_tmp_0 + 30] := S6[Slist_tmp_0];
END_FOR;
(* '<S1>:1:73' J = JacobianSpace(Slist_4DOF, thetalist0_4DOF); *)
(* *** CHAPTER 5: VELOCITY KINEMATICS AND STATICS *** *)
(* Takes Slist: The joint screw axes in the space frame when the manipulator *)
(* is at the home position, in the format of a matrix with the *)
(* screw axes as the columns, *)
(* thetalist: A list of joint coordinates.  *)
(* Returns the corresponding space Jacobian (6xn real numbers). *)
(* Example Input: *)
(* clear; clc; *)
(* Slist = [[0; 0; 1;   0; 0.2; 0.2], ... *)
(* [1; 0; 0;   2;   0;   3], ... *)
(* [0; 1; 0;   0;   2;   1], ... *)
(* [1; 0; 0; 0.2; 0.3; 0.4]]; *)
(* thetalist = [0.2; 1.1; 0.1; 1.2]; *)
(* Js = JacobianSpace(Slist, thetalist) *)
(* Output: *)
(* Js = *)
(* 0    0.9801   -0.0901    0.9575 *)
(* 0    0.1987    0.4446    0.2849 *)
(* 1.0000         0    0.8912   -0.0453 *)
(* 0    1.9522   -2.2164   -0.5116 *)
(* 0.2000    0.4365   -2.4371    2.7754 *)
(* 0.2000    2.9603    3.2357    2.2251 *)
(* 'JacobianSpace:27' Js = Slist; *)
(* MATLAB Function: '<Root>/MATLAB Function3' *)
FOR Slist_tmp_0 := 0 TO 35 DO 
    J[Slist_tmp_0] := Tsb_0[Slist_tmp_0];
END_FOR;
(* 'JacobianSpace:28' T = eye(4); *)
(* MATLAB Function: '<Root>/MATLAB Function3' *)
FOR Slist_tmp_0 := 0 TO 15 DO 
    T[Slist_tmp_0] := 0.0;
END_FOR;
T[0] := 1.0;
T[5] := 1.0;
T[10] := 1.0;
T[15] := 1.0;
(* 'JacobianSpace:29' for i = 2: length(thetalist) *)
(* MATLAB Function: '<Root>/MATLAB Function3' *)
se3mat[0] := 0.0;
se3mat[5] := 0.0;
se3mat[10] := 0.0;
se3mat[3] := 0.0;
se3mat[7] := 0.0;
se3mat[11] := 0.0;
se3mat[15] := 0.0;
(* MATLAB Function: '<Root>/MATLAB Function3' *)
tmp_0[0] := 0.0;
tmp_0[4] := 0.0;
tmp_0[8] := 0.0;
(* MATLAB Function: '<Root>/MATLAB Function3' *)
FOR b_i := 0 TO 4 DO 
    (* 'JacobianSpace:30' T = T * MatrixExp6(VecTose3(Slist(:, i - 1) * thetalist(i - 1))); *)
    thetalist0_0 := Vs[b_i];
    FOR Slist_tmp_0 := 0 TO 5 DO 
        V[Slist_tmp_0] := Tsb_0[(6 * b_i) + Slist_tmp_0] * thetalist0_0;
    END_FOR;
    (* *** CHAPTER 3: RIGID-BODY MOTIONS *** *)
    (* Takes a 6-vector (representing a spatial velocity). *)
    (* Returns the corresponding 4x4 se(3) matrix. *)
    (* Example Input: *)
    
    (* clear; clc; *)
    (* V = [1; 2; 3; 4; 5; 6]; *)
    (* se3mat = VecTose3(V) *)
    
    (* Output: *)
    (* se3mat = *)
    (* 0    -3     2     4 *)
    (* 3     0    -1     5 *)
    (* -2     1     0     6 *)
    (* 0     0     0     0  *)
    (* 'VecTose3:18' se3mat = [VecToso3(V(1: 3)), V(4: 6); 0, 0, 0, 0]; *)
    (* *** CHAPTER 3: RIGID-BODY MOTIONS *** *)
    (* Takes a 3-vector (angular velocity). *)
    (* Returns the skew symmetric matrix in so(3). *)
    (* Example Input: *)
    
    (* clear; clc; *)
    (* omg = [1; 2; 3]; *)
    (* so3mat = VecToso3(omg) *)
    
    (* Output: *)
    (* so3mat = *)
    (* 0    -3     2 *)
    (* 3     0    -1 *)
    (* -2     1     0 *)
    (* 'VecToso3:17' so3mat = [0, -omg(3), omg(2); omg(3), 0, -omg(1); -omg(2), omg(1), 0]; *)
    se3mat[4] :=  -V[2];
    se3mat[8] := V[1];
    se3mat[1] := V[2];
    se3mat[9] :=  -V[0];
    se3mat[2] :=  -V[1];
    se3mat[6] := V[0];
    se3mat[12] := V[3];
    se3mat[13] := V[4];
    se3mat[14] := V[5];
    (* *** CHAPTER 3: RIGID-BODY MOTIONS *** *)
    (* Takes a se(3) representation of exponential coordinates. *)
    (* Returns a T matrix in SE(3) that is achieved by traveling along/about the  *)
    (* screw axis S for a distance theta from an initial configuration T = I. *)
    (* Example Input: *)
    
    (* clear; clc; *)
    (* se3mat = [ 0,      0,       0,      0; *)
    (* 0,      0, -1.5708, 2.3562; *)
    (* 0, 1.5708,       0, 2.3562; *)
    (* 0,      0,       0,      0] *)
    (* T = MatrixExp6(se3mat) *)
    
    (* Output: *)
    (* T = *)
    (* 1.0000         0         0         0 *)
    (* 0    0.0000   -1.0000   -0.0000 *)
    (* 0    1.0000    0.0000    3.0000 *)
    (* 0         0         0    1.0000  *)
    (* 'MatrixExp6:22' omgtheta = so3ToVec(se3mat(1: 3, 1: 3)); *)
    (* *** CHAPTER 3: RIGID-BODY MOTIONS *** *)
    (* Takes a 3x3 skew-symmetric matrix (an element of so(3)). *)
    (* Returns the corresponding 3-vector (angular velocity). *)
    (* Example Input:  *)
    
    (* clear; clc; *)
    (* so3mat = [[0, -3, 2]; [3, 0, -1]; [-2, 1, 0]]; *)
    (* omg = so3ToVec(so3mat)   *)
    
    (* Output: *)
    (* omg = *)
    (* 1 *)
    (* 2 *)
    (* 3 *)
    (* 'so3ToVec:17' omg = [so3mat(3, 2); so3mat(1, 3); so3mat(2, 1)]; *)
    omgtheta[0] := V[0];
    omgtheta[1] := V[1];
    omgtheta[2] := V[2];
    (* 'MatrixExp6:23' if NearZero(norm(omgtheta)) *)
    (* *** BASIC HELPER FUNCTIONS *** *)
    (* Takes a scalar. *)
    (* Checks if the scalar is small enough to be neglected. *)
    (* Example Input: *)
    
    (* clear; clc; *)
    (* near = -1e-7; *)
    (* judge = NearZero(near) *)
    
    (* Output: *)
    (* judge = *)
    (* 1 *)
    (* 'NearZero:15' judge = norm(near) < 1e-6; *)
    c_theta := norm(x := omgtheta);
    IF ABS(c_theta) < 1.0E-6 THEN 
        (* 'MatrixExp6:24' T = [eye(3), se3mat(1: 3, 4); 0, 0, 0, 1]; *)
        i0_eye();
        tmp := i0_eye.I;
        FOR Slist_tmp_0 := 0 TO 2 DO 
            R_tmp := DWORD_TO_DINT(SHL(DINT_TO_DWORD(Slist_tmp_0), 2));
            a[R_tmp] := tmp[3 * Slist_tmp_0];
            a[R_tmp + 1] := tmp[(3 * Slist_tmp_0) + 1];
            a[R_tmp + 2] := tmp[(3 * Slist_tmp_0) + 2];
            a[Slist_tmp_0 + 12] := se3mat[Slist_tmp_0 + 12];
        END_FOR;
        a[3] := 0.0;
        a[7] := 0.0;
        a[11] := 0.0;
        a[15] := 1.0;
    ELSE 
        (* 'MatrixExp6:25' else *)
        (* 'MatrixExp6:26' [omghat, theta] = AxisAng3(omgtheta); *)
        (* *** CHAPTER 3: RIGID-BODY MOTIONS *** *)
        (* Takes A 3-vector of exponential coordinates for rotation. *)
        (* Returns the unit rotation axis omghat and the corresponding rotation  *)
        (* angle theta. *)
        (* Example Input: *)
        
        (* clear; clc; *)
        (* expc3 = [1; 2; 3]; *)
        (* [omghat, theta] = AxisAng3(expc3)   *)
        
        (* Output: *)
        (* omghat = *)
        (* 0.2673 *)
        (* 0.5345 *)
        (* 0.8018 *)
        (* theta = *)
        (* 3.7417 *)
        (* 'AxisAng3:20' theta = norm(expc3); *)
        (* 'AxisAng3:21' omghat = expc3 / theta; *)
        (* 'MatrixExp6:27' omgmat = se3mat(1: 3, 1: 3) / theta; *)
        FOR Slist_tmp_0 := 0 TO 2 DO 
            omgmat_tmp := DWORD_TO_DINT(SHL(DINT_TO_DWORD(Slist_tmp_0), 2));
            omgmat[3 * Slist_tmp_0] := se3mat[omgmat_tmp] / c_theta;
            omgmat[(3 * Slist_tmp_0) + 1] := se3mat[omgmat_tmp + 1] / c_theta;
            omgmat[(3 * Slist_tmp_0) + 2] := se3mat[omgmat_tmp + 2] / c_theta;
        END_FOR;
        (* 'MatrixExp6:28' T = [MatrixExp3(se3mat(1: 3, 1: 3)), ... *)
        (* 'MatrixExp6:29'          (eye(3) * theta + (1 - cos(theta)) * omgmat ... *)
        (* 'MatrixExp6:30'           + (theta - sin(theta)) * omgmat * omgmat) ... *)
        (* 'MatrixExp6:31'             * se3mat(1: 3, 4) / theta; *)
        (* 'MatrixExp6:32'          0, 0, 0, 1]; *)
        thetalist0_0 := 1.0 - COS(c_theta);
        g_a := c_theta - SIN(c_theta);
        (* *** CHAPTER 3: RIGID-BODY MOTIONS *** *)
        (* Takes a 3x3 so(3) representation of exponential coordinates. *)
        (* Returns R in SO(3) that is achieved by rotating about omghat by theta  *)
        (* from an initial orientation R = I. *)
        (* Example Input: *)
        
        (* clear; clc; *)
        (* so3mat = [[0, -3, 2]; [3, 0, -1]; [-2, 1, 0]]; *)
        (* R = MatrixExp3(so3mat)   *)
        
        (* Output: *)
        (* R = *)
        (* -0.6949    0.7135    0.0893 *)
        (* -0.1920   -0.3038    0.9332 *)
        (* 0.6930    0.6313    0.3481 *)
        (* 'MatrixExp3:18' omgtheta = so3ToVec(so3mat); *)
        (* *** CHAPTER 3: RIGID-BODY MOTIONS *** *)
        (* Takes a 3x3 skew-symmetric matrix (an element of so(3)). *)
        (* Returns the corresponding 3-vector (angular velocity). *)
        (* Example Input:  *)
        
        (* clear; clc; *)
        (* so3mat = [[0, -3, 2]; [3, 0, -1]; [-2, 1, 0]]; *)
        (* omg = so3ToVec(so3mat)   *)
        
        (* Output: *)
        (* omg = *)
        (* 1 *)
        (* 2 *)
        (* 3 *)
        (* 'so3ToVec:17' omg = [so3mat(3, 2); so3mat(1, 3); so3mat(2, 1)]; *)
        omgtheta[0] := V[0];
        omgtheta[1] := V[1];
        omgtheta[2] := V[2];
        (* 'MatrixExp3:19' if NearZero(norm(omgtheta)) *)
        (* *** BASIC HELPER FUNCTIONS *** *)
        (* Takes a scalar. *)
        (* Checks if the scalar is small enough to be neglected. *)
        (* Example Input: *)
        
        (* clear; clc; *)
        (* near = -1e-7; *)
        (* judge = NearZero(near) *)
        
        (* Output: *)
        (* judge = *)
        (* 1 *)
        (* 'NearZero:15' judge = norm(near) < 1e-6; *)
        i_theta := norm(x := omgtheta);
        IF ABS(i_theta) < 1.0E-6 THEN 
            (* 'MatrixExp3:20' R = eye(3); *)
            i0_eye();
            b_R := i0_eye.I;
        ELSE 
            (* 'MatrixExp3:21' else *)
            (* 'MatrixExp3:22' [omghat, theta] = AxisAng3(omgtheta); *)
            (* *** CHAPTER 3: RIGID-BODY MOTIONS *** *)
            (* Takes A 3-vector of exponential coordinates for rotation. *)
            (* Returns the unit rotation axis omghat and the corresponding rotation  *)
            (* angle theta. *)
            (* Example Input: *)
            
            (* clear; clc; *)
            (* expc3 = [1; 2; 3]; *)
            (* [omghat, theta] = AxisAng3(expc3)   *)
            
            (* Output: *)
            (* omghat = *)
            (* 0.2673 *)
            (* 0.5345 *)
            (* 0.8018 *)
            (* theta = *)
            (* 3.7417 *)
            (* 'AxisAng3:20' theta = norm(expc3); *)
            (* 'AxisAng3:21' omghat = expc3 / theta; *)
            (* 'MatrixExp3:23' omgmat = so3mat / theta; *)
            FOR Slist_tmp_0 := 0 TO 2 DO 
                omgmat_tmp := DWORD_TO_DINT(SHL(DINT_TO_DWORD(Slist_tmp_0), 2));
                b_omgmat[3 * Slist_tmp_0] := se3mat[omgmat_tmp] / i_theta;
                b_omgmat[(3 * Slist_tmp_0) + 1] := se3mat[omgmat_tmp + 1] / i_theta;
                b_omgmat[(3 * Slist_tmp_0) + 2] := se3mat[omgmat_tmp + 2] / i_theta;
            END_FOR;
            (* 'MatrixExp3:24' R = eye(3) + sin(theta) * omgmat + (1 - cos(theta)) * omgmat * omgmat; *)
            l_a := SIN(i_theta);
            x_tmp := COS(i_theta);
            i0_eye();
            tmp := i0_eye.I;
            FOR Slist_tmp_0 := 0 TO 2 DO 
                FOR omgmat_tmp := 0 TO 2 DO 
                    R_tmp := (3 * omgmat_tmp) + Slist_tmp_0;
                    b_R[R_tmp] := (((((1.0 - x_tmp) * b_omgmat[Slist_tmp_0 + 3]) * b_omgmat[(3 * omgmat_tmp) + 1]) + (((1.0 - x_tmp) * b_omgmat[Slist_tmp_0]) * b_omgmat[3 * omgmat_tmp])) + ((b_omgmat[Slist_tmp_0 + 6] * (1.0 - x_tmp)) * b_omgmat[(3 * omgmat_tmp) + 2])) + ((b_omgmat[R_tmp] * l_a) + tmp[R_tmp]);
                END_FOR;
            END_FOR;
        END_IF;
        FOR Slist_tmp_0 := 0 TO 2 DO 
            l_a := 0.0;
            FOR omgmat_tmp := 0 TO 2 DO 
                R_tmp := (3 * omgmat_tmp) + Slist_tmp_0;
                l_a := ((((((omgmat[Slist_tmp_0 + 3] * g_a) * omgmat[(3 * omgmat_tmp) + 1]) + ((g_a * omgmat[Slist_tmp_0]) * omgmat[3 * omgmat_tmp])) + ((omgmat[Slist_tmp_0 + 6] * g_a) * omgmat[(3 * omgmat_tmp) + 2])) + ((SINT_TO_LREAL(p_a[R_tmp]) * c_theta) + (omgmat[R_tmp] * thetalist0_0))) * se3mat[omgmat_tmp + 12]) + l_a;
                a[omgmat_tmp + (Slist_tmp_0 * 4)] := b_R[(3 * Slist_tmp_0) + omgmat_tmp];
            END_FOR;
            a[Slist_tmp_0 + 12] := l_a / c_theta;
        END_FOR;
        a[3] := 0.0;
        a[7] := 0.0;
        a[11] := 0.0;
        a[15] := 1.0;
    END_IF;
    FOR Slist_tmp_0 := 0 TO 3 DO 
        FOR omgmat_tmp := 0 TO 3 DO 
            R_tmp := DWORD_TO_DINT(SHL(DINT_TO_DWORD(omgmat_tmp), 2));
            i := Slist_tmp_0 + R_tmp;
            M[i] := 0.0;
            M[i] := M[i] + (a[R_tmp] * T[Slist_tmp_0]);
            M[i] := (a[R_tmp + 1] * T[Slist_tmp_0 + 4]) + M[i];
            M[i] := (a[R_tmp + 2] * T[Slist_tmp_0 + 8]) + M[i];
            M[i] := (a[R_tmp + 3] * T[Slist_tmp_0 + 12]) + M[i];
        END_FOR;
    END_FOR;
    FOR Slist_tmp_0 := 0 TO 15 DO 
        T[Slist_tmp_0] := M[Slist_tmp_0];
    END_FOR;
    (* 'JacobianSpace:31' Js(:, i) = Adjoint(T) * Slist(:, i); *)
    (* *** CHAPTER 3: RIGID-BODY MOTIONS *** *)
    (* Takes T a transformation matrix SE3.  *)
    (* Returns the corresponding 6x6 adjoint representation [AdT]. *)
    (* Example Input: *)
    
    (* clear; clc; *)
    (* T = [[1, 0, 0, 0]; [0, 0, -1, 0]; [0, 1, 0, 3]; [0, 0, 0, 1]]; *)
    (* AdT = Adjoint(T) *)
    
    (* Output: *)
    (* AdT = *)
    (* 1     0     0     0     0     0 *)
    (* 0     0    -1     0     0     0 *)
    (* 0     1     0     0     0     0 *)
    (* 0     0     3     1     0     0 *)
    (* 3     0     0     0     0    -1 *)
    (* 0     0     0     0     1     0 *)
    (* 'Adjoint:20' [R, p] = TransToRp(T); *)
    (* *** CHAPTER 3: RIGID-BODY MOTIONS *** *)
    (* Takes the transformation matrix T in SE(3)  *)
    (* Returns R: the corresponding rotation matrix *)
    (* p: the corresponding position vector . *)
    (* Example Input: *)
    
    (* clear; clc; *)
    (* T = [[1, 0, 0, 0]; [0, 0, -1, 0]; [0, 1, 0, 3]; [0, 0, 0, 1]]; *)
    (* [R, p] = TransToRp(T) *)
    
    (* Output: *)
    (* R = *)
    (* 1     0     0 *)
    (* 0     0    -1 *)
    (* 0     1     0 *)
    (* p = *)
    (* 0 *)
    (* 0 *)
    (* 3 *)
    (* 'TransToRp:22' R = T(1: 3, 1: 3); *)
    (* 'TransToRp:23' p = T(1: 3, 4); *)
    (* 'Adjoint:21' AdT = [R, zeros(3); VecToso3(p) * R, R]; *)
    (* *** CHAPTER 3: RIGID-BODY MOTIONS *** *)
    (* Takes a 3-vector (angular velocity). *)
    (* Returns the skew symmetric matrix in so(3). *)
    (* Example Input: *)
    
    (* clear; clc; *)
    (* omg = [1; 2; 3]; *)
    (* so3mat = VecToso3(omg) *)
    
    (* Output: *)
    (* so3mat = *)
    (* 0    -3     2 *)
    (* 3     0    -1 *)
    (* -2     1     0 *)
    (* 'VecToso3:17' so3mat = [0, -omg(3), omg(2); omg(3), 0, -omg(1); -omg(2), omg(1), 0]; *)
    tmp_0[3] :=  -T[14];
    tmp_0[6] := T[13];
    tmp_0[1] := T[14];
    tmp_0[7] :=  -T[12];
    tmp_0[2] :=  -T[13];
    tmp_0[5] := T[12];
    FOR Slist_tmp_0 := 0 TO 2 DO 
        FOR omgmat_tmp := 0 TO 2 DO 
            R_tmp := Slist_tmp_0 + (3 * omgmat_tmp);
            tmp[R_tmp] := 0.0;
            a_tmp_tmp := DWORD_TO_DINT(SHL(DINT_TO_DWORD(omgmat_tmp), 2));
            tmp[R_tmp] := tmp[R_tmp] + (T[a_tmp_tmp] * tmp_0[Slist_tmp_0]);
            tmp[R_tmp] := (T[a_tmp_tmp + 1] * tmp_0[Slist_tmp_0 + 3]) + tmp[R_tmp];
            tmp[R_tmp] := (T[a_tmp_tmp + 2] * tmp_0[Slist_tmp_0 + 6]) + tmp[R_tmp];
            T_0[omgmat_tmp + (6 * Slist_tmp_0)] := T[(Slist_tmp_0 * 4) + omgmat_tmp];
            T_0[omgmat_tmp + (6 * (Slist_tmp_0 + 3))] := 0.0;
        END_FOR;
    END_FOR;
    FOR Slist_tmp_0 := 0 TO 2 DO 
        T_0[(6 * Slist_tmp_0) + 3] := tmp[3 * Slist_tmp_0];
        i := DWORD_TO_DINT(SHL(DINT_TO_DWORD(Slist_tmp_0), 2));
        omgmat_tmp := 6 * (Slist_tmp_0 + 3);
        T_0[omgmat_tmp + 3] := T[i];
        T_0[(6 * Slist_tmp_0) + 4] := tmp[(3 * Slist_tmp_0) + 1];
        T_0[omgmat_tmp + 4] := T[i + 1];
        T_0[(6 * Slist_tmp_0) + 5] := tmp[(3 * Slist_tmp_0) + 2];
        T_0[omgmat_tmp + 5] := T[i + 2];
    END_FOR;
    FOR Slist_tmp_0 := 0 TO 5 DO 
        i := 6 * (b_i + 1);
        R_tmp := Slist_tmp_0 + i;
        J[R_tmp] := 0.0;
        FOR omgmat_tmp := 0 TO 5 DO 
            J[R_tmp] := (Tsb_0[i + omgmat_tmp] * T_0[(6 * omgmat_tmp) + Slist_tmp_0]) + J[R_tmp];
        END_FOR;
    END_FOR;
END_FOR;
(* Outport: '<Root>/q1' incorporates:
 *  MATLAB Function: '<Root>/MATLAB Function3' *)
(* '<S1>:1:74' thetalistDot = pinv(J) * Vs; *)
(* '<S1>:1:76' q1 = thetalist(1); *)
(* '<S1>:1:77' q2 = thetalist(2); *)
(* '<S1>:1:78' q3 = thetalist(3); *)
(* '<S1>:1:79' q4Dot = thetalistDot(4); *)
q1 := thetalist0[0];
(* Outport: '<Root>/q2' incorporates:
 *  MATLAB Function: '<Root>/MATLAB Function3' *)
q2 := thetalist0[1];
(* Outport: '<Root>/q3' incorporates:
 *  MATLAB Function: '<Root>/MATLAB Function3' *)
q3 := thetalist0[2];
(* MATLAB Function: '<Root>/MATLAB Function3' *)
i0_pinv_i(A := J);
Tsb_0 := i0_pinv_i.X;
(* MATLAB Function: '<Root>/MATLAB Function3' *)
V[0] := 0.0;
V[1] := 0.0;
V[2] := 0.0;
V[3] := Vx;
V[4] := Vy;
V[5] := Vz;
(* MATLAB Function: '<Root>/MATLAB Function3' *)
FOR Slist_tmp_0 := 0 TO 5 DO 
    tmp_2[Slist_tmp_0] := 0.0;
    FOR omgmat_tmp := 0 TO 5 DO 
        tmp_2[Slist_tmp_0] := (Tsb_0[(6 * omgmat_tmp) + Slist_tmp_0] * V[omgmat_tmp]) + tmp_2[Slist_tmp_0];
    END_FOR;
END_FOR;
(* Outport: '<Root>/q4Dot' incorporates:
 *  MATLAB Function: '<Root>/MATLAB Function3' *)
q4Dot := tmp_2[3];
(* Outport: '<Root>/success' incorporates:
 *  MATLAB Function: '<Root>/MATLAB Function3' *)
success :=  NOT err;

END_FUNCTION_BLOCK

// ---- KinematicsForwAndInverseMatLab/MatrixLog3.TcPOU
FUNCTION_BLOCK MatrixLog3
VAR_INPUT
    b_R: ARRAY [0..8] OF LREAL;
END_VAR
VAR_OUTPUT
    so3mat: ARRAY [0..8] OF LREAL;
END_VAR
VAR_TEMP
    acosinput: LREAL;
    theta: LREAL;
    t: LREAL;
    i: DINT;
    b_idx_0: LREAL;
    b_idx_1: LREAL;
    so3mat_tmp: DINT;
END_VAR

(* 'MatrixLog3:18' acosinput = (trace(R) - 1) / 2; *)
acosinput := (((b_R[0] + b_R[4]) + b_R[8]) - 1.0) / 2.0;
(* 'MatrixLog3:19' if acosinput >= 1 *)
IF acosinput >= 1.0 THEN 
    (* 'MatrixLog3:20' so3mat = zeros(3); *)
    FOR i := 0 TO 8 DO 
        so3mat[i] := 0.0;
    END_FOR;
ELSIF acosinput <= -1.0 THEN 
    (* 'MatrixLog3:21' elseif acosinput <= -1 *)
    (* 'MatrixLog3:22' if ~NearZero(1 + R(3, 3)) *)
    (* *** BASIC HELPER FUNCTIONS *** *)
    (* Takes a scalar. *)
    (* Checks if the scalar is small enough to be neglected. *)
    (* Example Input: *)
    
    (* clear; clc; *)
    (* near = -1e-7; *)
    (* judge = NearZero(near) *)
    
    (* Output: *)
    (* judge = *)
    (* 1 *)
    (* 'NearZero:15' judge = norm(near) < 1e-6; *)
    IF ABS(b_R[8] + 1.0) >= 1.0E-6 THEN 
        (* 'MatrixLog3:23' omg = (1 / sqrt(2 * (1 + R(3, 3)))) ... *)
        (* 'MatrixLog3:24'               * [R(1, 3); R(2, 3); 1 + R(3, 3)]; *)
        t := 1.0 / SQRT((b_R[8] + 1.0) * 2.0);
        b_idx_0 := t * b_R[6];
        b_idx_1 := t * b_R[7];
        t := (b_R[8] + 1.0) * t;
    ELSE 
        (* *** BASIC HELPER FUNCTIONS *** *)
        (* Takes a scalar. *)
        (* Checks if the scalar is small enough to be neglected. *)
        (* Example Input: *)
        
        (* clear; clc; *)
        (* near = -1e-7; *)
        (* judge = NearZero(near) *)
        
        (* Output: *)
        (* judge = *)
        (* 1 *)
        (* 'NearZero:15' judge = norm(near) < 1e-6; *)
        IF ABS(b_R[4] + 1.0) >= 1.0E-6 THEN 
            (* 'MatrixLog3:25' elseif ~NearZero(1 + R(2, 2)) *)
            (* 'MatrixLog3:26' omg = (1 / sqrt(2 * (1 + R(2, 2)))) ... *)
            (* 'MatrixLog3:27'               * [R(1, 2); 1 + R(2, 2); R(3, 2)]; *)
            t := 1.0 / SQRT((b_R[4] + 1.0) * 2.0);
            b_idx_0 := t * b_R[3];
            b_idx_1 := (b_R[4] + 1.0) * t;
            t := t * b_R[5];
        ELSE 
            (* 'MatrixLog3:28' else *)
            (* 'MatrixLog3:29' omg = (1 / sqrt(2 * (1 + R(1, 1)))) ... *)
            (* 'MatrixLog3:30'               * [1 + R(1, 1); R(2, 1); R(3, 1)]; *)
            t := 1.0 / SQRT((b_R[0] + 1.0) * 2.0);
            b_idx_0 := (b_R[0] + 1.0) * t;
            b_idx_1 := t * b_R[1];
            t := t * b_R[2];
        END_IF;
    END_IF;
    (* 'MatrixLog3:32' so3mat = VecToso3(pi * omg); *)
    b_idx_0 := 3.1415926535897931 * b_idx_0;
    b_idx_1 := 3.1415926535897931 * b_idx_1;
    t := 3.1415926535897931 * t;
    (* *** CHAPTER 3: RIGID-BODY MOTIONS *** *)
    (* Takes a 3-vector (angular velocity). *)
    (* Returns the skew symmetric matrix in so(3). *)
    (* Example Input: *)
    
    (* clear; clc; *)
    (* omg = [1; 2; 3]; *)
    (* so3mat = VecToso3(omg) *)
    
    (* Output: *)
    (* so3mat = *)
    (* 0    -3     2 *)
    (* 3     0    -1 *)
    (* -2     1     0 *)
    (* 'VecToso3:17' so3mat = [0, -omg(3), omg(2); omg(3), 0, -omg(1); -omg(2), omg(1), 0]; *)
    so3mat[0] := 0.0;
    so3mat[3] :=  -t;
    so3mat[6] := b_idx_1;
    so3mat[1] := t;
    so3mat[4] := 0.0;
    so3mat[7] :=  -b_idx_0;
    so3mat[2] :=  -b_idx_1;
    so3mat[5] := b_idx_0;
    so3mat[8] := 0.0;
ELSE 
    (* 'MatrixLog3:33' else *)
    (* 'MatrixLog3:34' theta = acos(acosinput); *)
    theta := ACOS(acosinput);
    (* 'MatrixLog3:35' so3mat = theta * (1 / (2 * sin(theta))) * (R - R'); *)
    t := (1.0 / (2.0 * SIN(theta))) * theta;
    FOR i := 0 TO 2 DO 
        so3mat[3 * i] := (b_R[3 * i] - b_R[i]) * t;
        so3mat_tmp := (3 * i) + 1;
        so3mat[so3mat_tmp] := (b_R[so3mat_tmp] - b_R[i + 3]) * t;
        so3mat_tmp := (3 * i) + 2;
        so3mat[so3mat_tmp] := (b_R[so3mat_tmp] - b_R[i + 6]) * t;
    END_FOR;
END_IF;

END_FUNCTION_BLOCK

// ---- KinematicsForwAndInverseMatLab/eye.TcPOU
FUNCTION_BLOCK eye
VAR_OUTPUT
    I: ARRAY [0..8] OF LREAL;
END_VAR
VAR_TEMP
    b_i: DINT;
END_VAR

FOR b_i := 0 TO 8 DO 
    I[b_i] := 0.0;
END_FOR;
I[0] := 1.0;
I[4] := 1.0;
I[8] := 1.0;

END_FUNCTION_BLOCK

// ---- KinematicsForwAndInverseMatLab/pinv.TcPOU
FUNCTION_BLOCK pinv
VAR_INPUT
    A: ARRAY [0..29] OF LREAL;
END_VAR
VAR_OUTPUT
    X: ARRAY [0..29] OF LREAL;
END_VAR
VAR
    i0_svd: svd;
END_VAR
VAR_TEMP
    V: ARRAY [0..24] OF LREAL;
    b_r: DINT;
    vcol: DINT;
    U: ARRAY [0..29] OF LREAL;
    b_s: ARRAY [0..4] OF LREAL;
    tol: LREAL;
    j: DINT;
    ar: DINT;
    ia: DINT;
    b: DINT;
    ib: DINT;
    b_ic: DINT;
    exitg1: DINT;
END_VAR

b_r := -1;
FOR vcol := 0 TO 29 DO 
    X[vcol] := 0.0;
END_FOR;
i0_svd(A := A);
U := i0_svd.U;
b_s := i0_svd.b_s;
V := i0_svd.V;
tol := 6.0 * eps(x := b_s[0]);
vcol := 0;
REPEAT 
    exitg1 := 0;
    IF vcol < 5 THEN 
        IF b_s[vcol] <= tol THEN 
            exitg1 := 1;
        ELSE 
            b_r := b_r + 1;
            vcol := vcol + 1;
        END_IF;
    ELSE 
        exitg1 := 1;
    END_IF;
UNTIL NOT(exitg1 = 0)
END_REPEAT;
IF (b_r + 1) > 0 THEN 
    vcol := 0;
    j := 0;
    WHILE j <= b_r DO
        tol := 1.0 / b_s[j];
        ar := vcol;
        WHILE (ar + 1) <= (vcol + 5) DO
            V[ar] := tol * V[ar];
            ar := ar + 1;
        END_WHILE;
        vcol := vcol + 5;
        j := j + 1;
    END_WHILE;
    vcol := 0;
    FOR j := 0 TO 26 BY 5 DO 
        ar := j;
        WHILE (ar + 1) <= (j + 5) DO
            X[ar] := 0.0;
            ar := ar + 1;
        END_WHILE;
    END_FOR;
    FOR j := 0 TO 26 BY 5 DO 
        ar := -1;
        vcol := vcol + 1;
        b := (6 * b_r) + vcol;
        ib := vcol;
        WHILE ib <= b DO
            ia := ar;
            b_ic := j;
            WHILE (b_ic + 1) <= (j + 5) DO
                ia := ia + 1;
                X[b_ic] := (U[ib - 1] * V[ia]) + X[b_ic];
                b_ic := b_ic + 1;
            END_WHILE;
            ar := ar + 5;
            ib := ib + 6;
        END_WHILE;
    END_FOR;
END_IF;

END_FUNCTION_BLOCK

// ---- KinematicsForwAndInverseMatLab/svd.TcPOU
FUNCTION_BLOCK svd
VAR_INPUT
    A: ARRAY [0..29] OF LREAL;
END_VAR
VAR_OUTPUT
    U: ARRAY [0..29] OF LREAL;
    b_s: ARRAY [0..4] OF LREAL;
    V: ARRAY [0..24] OF LREAL;
END_VAR
VAR
    i0_xrot_c: xrot_c;
    i0_xrotg: xrotg;
    i0_xrot: xrot;
    i0_xswap_g: xswap_g;
    i0_xswap: xswap;
    i0_xscal_fiz: xscal_fiz;
    i0_xscal_fi: xscal_fi;
    i0_xaxpy_dmy: xaxpy_dmy;
    i0_xaxpy: xaxpy;
    i0_xaxpy_d: xaxpy_d;
    i0_xaxpy_dm: xaxpy_dm;
    i0_xscal_f: xscal_f;
    i0_xscal: xscal;
END_VAR
VAR_TEMP
    b_A: ARRAY [0..29] OF LREAL;
    b_b_s: ARRAY [0..4] OF LREAL;
    e: ARRAY [0..4] OF LREAL;
    work: ARRAY [0..5] OF LREAL;
    Vf: ARRAY [0..24] OF LREAL;
    qq: DINT;
    apply_transform: BOOL;
    nrm: LREAL;
    qjj: DINT;
    qp1jj: DINT;
    m: DINT;
    qp1q: DINT;
    rt: LREAL;
    ztest: LREAL;
    smm1: LREAL;
    emm1: LREAL;
    sqds: LREAL;
    shift: LREAL;
    j_ii: DINT;
    exitg1: DINT;
    temp1: LREAL;
    temp2: LREAL;
    temp3: LREAL;
    temp4: LREAL;
    temp5: LREAL;
    temp6: LREAL;
    temp7: LREAL;
    temp8: LREAL;
    temp9: LREAL;
    temp10: LREAL;
    temp11: LREAL;
    temp12: LREAL;
    temp13: LREAL;
    temp14: LREAL;
END_VAR

FOR m := 0 TO 29 DO 
    b_A[m] := A[m];
END_FOR;
FOR m := 0 TO 4 DO 
    b_b_s[m] := 0.0;
    e[m] := 0.0;
END_FOR;
FOR m := 0 TO 5 DO 
    work[m] := 0.0;
END_FOR;
FOR m := 0 TO 29 DO 
    U[m] := 0.0;
END_FOR;
FOR m := 0 TO 24 DO 
    Vf[m] := 0.0;
END_FOR;
FOR m := 0 TO 4 DO 
    qq := (6 * m) + m;
    apply_transform := FALSE;
    nrm := xnrm2(b_n := 6 - m, x := b_A, ix0 := qq + 1);
    IF nrm > 0.0 THEN 
        apply_transform := TRUE;
        IF b_A[qq] < 0.0 THEN 
            b_b_s[m] :=  -nrm;
        ELSE 
            b_b_s[m] := nrm;
        END_IF;
        IF ABS(b_b_s[m]) >= 1.0020841800044864E-292 THEN 
            i0_xscal(b_n := 6 - m, a := 1.0 / b_b_s[m], x := b_A, ix0 := qq + 1);
        ELSE 
            qp1q := (qq - m) + 6;
            qjj := qq;
            WHILE (qjj + 1) <= qp1q DO
                b_A[qjj] := b_A[qjj] / b_b_s[m];
                qjj := qjj + 1;
            END_WHILE;
        END_IF;
        b_A[qq] := b_A[qq] + 1.0;
        b_b_s[m] :=  -b_b_s[m];
    ELSE 
        b_b_s[m] := 0.0;
    END_IF;
    qp1q := m + 1;
    WHILE (qp1q + 1) < 6 DO
        qjj := (6 * qp1q) + m;
        IF apply_transform THEN 
            temp1 := xdotc(b_n := 6 - m, x := b_A, ix0 := qq + 1, y := b_A, iy0 := qjj + 1);
            i0_xaxpy(b_n := 6 - m, a :=  -(temp1 / b_A[m + (6 * m)]), ix0 := qq + 1, y := b_A, iy0 := qjj + 1);
        END_IF;
        e[qp1q] := b_A[qjj];
        qp1q := qp1q + 1;
    END_WHILE;
    qq := m;
    WHILE (qq + 1) < 7 DO
        U[qq + (6 * m)] := b_A[(6 * m) + qq];
        qq := qq + 1;
    END_WHILE;
    IF (m + 1) <= 3 THEN 
        nrm := xnrm2_l(b_n := 4 - m, x := e, ix0 := m + 2);
        IF nrm = 0.0 THEN 
            e[m] := 0.0;
        ELSE 
            IF e[m + 1] < 0.0 THEN 
                e[m] :=  -nrm;
            ELSE 
                e[m] := nrm;
            END_IF;
            nrm := e[m];
            IF ABS(e[m]) >= 1.0020841800044864E-292 THEN 
                i0_xscal_f(b_n := 4 - m, a := 1.0 / e[m], x := e, ix0 := m + 2);
            ELSE 
                qq := m + 1;
                WHILE (qq + 1) <= 5 DO
                    e[qq] := e[qq] / nrm;
                    qq := qq + 1;
                END_WHILE;
            END_IF;
            e[m + 1] := e[m + 1] + 1.0;
            e[m] :=  -e[m];
            qq := m + 1;
            WHILE (qq + 1) < 7 DO
                work[qq] := 0.0;
                qq := qq + 1;
            END_WHILE;
            qq := m + 1;
            WHILE (qq + 1) < 6 DO
                i0_xaxpy_d(b_n := 5 - m, a := e[qq], x := b_A, ix0 := (m + (6 * qq)) + 2, y := work, iy0 := m + 2);
                qq := qq + 1;
            END_WHILE;
            qq := m + 1;
            WHILE (qq + 1) < 6 DO
                i0_xaxpy_dm(b_n := 5 - m, a := ( -e[qq]) / e[m + 1], x := work, ix0 := m + 2, y := b_A, iy0 := (m + (6 * qq)) + 2);
                qq := qq + 1;
            END_WHILE;
        END_IF;
        qq := m + 1;
        WHILE (qq + 1) < 6 DO
            Vf[qq + (5 * m)] := e[qq];
            qq := qq + 1;
        END_WHILE;
    END_IF;
END_FOR;
m := 3;
e[3] := b_A[27];
e[4] := 0.0;
FOR qp1q := 4 TO 0 BY -1 DO 
    qq := (6 * qp1q) + qp1q;
    IF b_b_s[qp1q] <> 0.0 THEN 
        qp1jj := qp1q + 1;
        WHILE (qp1jj + 1) < 6 DO
            qjj := ((6 * qp1jj) + qp1q) + 1;
            temp2 := xdotc(b_n := 6 - qp1q, x := U, ix0 := qq + 1, y := U, iy0 := qjj);
            i0_xaxpy(b_n := 6 - qp1q, a :=  -(temp2 / U[qq]), ix0 := qq + 1, y := U, iy0 := qjj);
            qp1jj := qp1jj + 1;
        END_WHILE;
        qjj := qp1q;
        WHILE (qjj + 1) < 7 DO
            qp1jj := (6 * qp1q) + qjj;
            U[qp1jj] :=  -U[qp1jj];
            qjj := qjj + 1;
        END_WHILE;
        U[qq] := U[qq] + 1.0;
        qq := 0;
        WHILE qq <= (qp1q - 1) DO
            U[qq + (6 * qp1q)] := 0.0;
            qq := qq + 1;
        END_WHILE;
    ELSE 
        FOR qjj := 0 TO 5 DO 
            U[qjj + (6 * qp1q)] := 0.0;
        END_FOR;
        U[qq] := 1.0;
    END_IF;
END_FOR;
FOR qq := 4 TO 0 BY -1 DO 
    IF (qq + 1) <= 3 THEN 
        IF e[qq] <> 0.0 THEN 
            qp1q := ((5 * qq) + qq) + 2;
            qjj := qq + 1;
            WHILE (qjj + 1) < 6 DO
                qp1jj := ((5 * qjj) + qq) + 2;
                temp3 := xdotc_i(b_n := 4 - qq, x := Vf, ix0 := qp1q, y := Vf, iy0 := qp1jj);
                i0_xaxpy_dmy(b_n := 4 - qq, a :=  -(temp3 / Vf[qp1q - 1]), ix0 := qp1q, y := Vf, iy0 := qp1jj);
                qjj := qjj + 1;
            END_WHILE;
        END_IF;
    END_IF;
    FOR qp1q := 0 TO 4 DO 
        Vf[qp1q + (5 * qq)] := 0.0;
    END_FOR;
    Vf[qq + (5 * qq)] := 1.0;
END_FOR;
FOR qq := 0 TO 4 DO 
    ztest := e[qq];
    IF b_b_s[qq] <> 0.0 THEN 
        rt := ABS(b_b_s[qq]);
        nrm := b_b_s[qq] / rt;
        b_b_s[qq] := rt;
        IF (qq + 1) < 5 THEN 
            ztest := ztest / nrm;
        END_IF;
        i0_xscal_fi(a := nrm, x := U, ix0 := (6 * qq) + 1);
    END_IF;
    IF (qq + 1) < 5 THEN 
        IF ztest <> 0.0 THEN 
            rt := ABS(ztest);
            nrm := rt / ztest;
            ztest := rt;
            b_b_s[qq + 1] := b_b_s[qq + 1] * nrm;
            i0_xscal_fiz(a := nrm, x := Vf, ix0 := (5 * (qq + 1)) + 1);
        END_IF;
    END_IF;
    e[qq] := ztest;
END_FOR;
qq := 0;
nrm := 0.0;
FOR qp1q := 0 TO 4 DO 
    temp4 := ABS(b_b_s[qp1q]);
    temp5 := ABS(e[qp1q]);
    temp6 := MAX(temp4, temp5);
    nrm := MAX(nrm, temp6);
END_FOR;
WHILE ((m + 2) > 0) AND (qq < 75) DO
    qp1jj := m + 1;
    REPEAT 
        exitg1 := 0;
        qp1q := qp1jj;
        IF qp1jj = 0 THEN 
            exitg1 := 1;
        ELSE 
            rt := ABS(e[qp1jj - 1]);
            IF rt <= ((ABS(b_b_s[qp1jj - 1]) + ABS(b_b_s[qp1jj])) * 2.2204460492503131E-16) THEN 
                e[qp1jj - 1] := 0.0;
                exitg1 := 1;
            ELSIF (rt <= 1.0020841800044864E-292) OR ((qq > 20) AND (rt <= (2.2204460492503131E-16 * nrm))) THEN 
                e[qp1jj - 1] := 0.0;
                exitg1 := 1;
            ELSE 
                qp1jj := qp1jj - 1;
            END_IF;
        END_IF;
    UNTIL NOT(exitg1 = 0)
    END_REPEAT;
    IF (m + 1) = qp1jj THEN 
        qp1jj := 4;
    ELSE 
        qjj := m + 2;
        j_ii := m + 2;
        REPEAT 
            exitg1 := 0;
            IF j_ii >= qp1jj THEN 
                qjj := j_ii;
                IF j_ii = qp1jj THEN 
                    exitg1 := 1;
                ELSE 
                    rt := 0.0;
                    IF j_ii < (m + 2) THEN 
                        rt := ABS(e[j_ii - 1]);
                    END_IF;
                    IF j_ii > (qp1jj + 1) THEN 
                        rt := ABS(e[j_ii - 2]) + rt;
                    END_IF;
                    ztest := ABS(b_b_s[j_ii - 1]);
                    IF (ztest <= (2.2204460492503131E-16 * rt)) OR (ztest <= 1.0020841800044864E-292) THEN 
                        b_b_s[j_ii - 1] := 0.0;
                        exitg1 := 1;
                    ELSE 
                        j_ii := j_ii - 1;
                    END_IF;
                END_IF;
            ELSE 
                exitg1 := 1;
            END_IF;
        UNTIL NOT(exitg1 = 0)
        END_REPEAT;
        IF qjj = qp1jj THEN 
            qp1jj := 3;
        ELSIF (m + 2) = qjj THEN 
            qp1jj := 1;
        ELSE 
            qp1jj := 2;
            qp1q := qjj;
        END_IF;
    END_IF;
    CASE qp1jj OF
        1: 
            rt := e[m];
            e[m] := 0.0;
            qjj := m;
            WHILE (qjj + 1) >= (qp1q + 1) DO
                i0_xrotg(a := b_b_s[qjj], b := rt);
                ztest := i0_xrotg.c;
                sqds := i0_xrotg.b_s;
                IF (qjj + 1) > (qp1q + 1) THEN 
                    emm1 := e[qjj - 1];
                    rt := emm1 * ( -sqds);
                    e[qjj - 1] := emm1 * ztest;
                END_IF;
                i0_xrot(x := Vf, ix0 := (5 * qjj) + 1, iy0 := (5 * (m + 1)) + 1, c := ztest, b_s := sqds);
                qjj := qjj - 1;
            END_WHILE;
        2: 
            rt := e[qp1q - 1];
            e[qp1q - 1] := 0.0;
            qjj := qp1q;
            WHILE (qjj + 1) <= (m + 2) DO
                i0_xrotg(a := b_b_s[qjj], b := rt);
                ztest := i0_xrotg.c;
                sqds := i0_xrotg.b_s;
                rt := ( -sqds) * e[qjj];
                e[qjj] := e[qjj] * ztest;
                i0_xrot_c(x := U, ix0 := (6 * qjj) + 1, iy0 := (6 * (qp1q - 1)) + 1, c := ztest, b_s := sqds);
                qjj := qjj + 1;
            END_WHILE;
        3: 
            rt := b_b_s[m + 1];
            temp7 := ABS(rt);
            temp8 := ABS(b_b_s[m]);
            temp9 := MAX(temp7, temp8);
            temp10 := ABS(e[m]);
            temp11 := MAX(temp9, temp10);
            temp12 := ABS(b_b_s[qp1q]);
            temp13 := MAX(temp11, temp12);
            temp14 := ABS(e[qp1q]);
            ztest := MAX(temp13, temp14);
            rt := rt / ztest;
            smm1 := b_b_s[m] / ztest;
            emm1 := e[m] / ztest;
            sqds := b_b_s[qp1q] / ztest;
            smm1 := (((smm1 + rt) * (smm1 - rt)) + (emm1 * emm1)) / 2.0;
            emm1 := rt * emm1;
            emm1 := emm1 * emm1;
            IF (smm1 <> 0.0) OR (emm1 <> 0.0) THEN 
                shift := SQRT((smm1 * smm1) + emm1);
                IF smm1 < 0.0 THEN 
                    shift :=  -shift;
                END_IF;
                shift := emm1 / (smm1 + shift);
            ELSE 
                shift := 0.0;
            END_IF;
            rt := ((sqds + rt) * (sqds - rt)) + shift;
            ztest := (e[qp1q] / ztest) * sqds;
            qjj := qp1q + 1;
            WHILE qjj <= (m + 1) DO
                i0_xrotg(a := rt, b := ztest);
                sqds := i0_xrotg.c;
                smm1 := i0_xrotg.b_s;
                IF qjj > (qp1q + 1) THEN 
                    e[qjj - 2] := rt;
                END_IF;
                emm1 := e[qjj - 1];
                rt := b_b_s[qjj - 1];
                e[qjj - 1] := (emm1 * sqds) - (rt * smm1);
                ztest := smm1 * b_b_s[qjj];
                b_b_s[qjj] := b_b_s[qjj] * sqds;
                i0_xrot(x := Vf, ix0 := (5 * (qjj - 1)) + 1, iy0 := (5 * qjj) + 1, c := sqds, b_s := smm1);
                b_b_s[qjj - 1] := (rt * sqds) + (emm1 * smm1);
                i0_xrotg(a := b_b_s[qjj - 1], b := ztest);
                sqds := i0_xrotg.c;
                smm1 := i0_xrotg.b_s;
                rt := (e[qjj - 1] * sqds) + (smm1 * b_b_s[qjj]);
                b_b_s[qjj] := (e[qjj - 1] * ( -smm1)) + (sqds * b_b_s[qjj]);
                ztest := smm1 * e[qjj];
                e[qjj] := e[qjj] * sqds;
                i0_xrot_c(x := U, ix0 := (6 * (qjj - 1)) + 1, iy0 := (6 * qjj) + 1, c := sqds, b_s := smm1);
                qjj := qjj + 1;
            END_WHILE;
            e[m] := rt;
            qq := qq + 1;
        ELSE
            IF b_b_s[qp1q] < 0.0 THEN 
                b_b_s[qp1q] :=  -b_b_s[qp1q];
                i0_xscal_fiz(a := -1.0, x := Vf, ix0 := (5 * qp1q) + 1);
            END_IF;
            qq := qp1q + 1;
            REPEAT 
                exitg1 := 0;
                IF (qp1q + 1) < 5 THEN 
                    IF b_b_s[qp1q] < b_b_s[qq] THEN 
                        rt := b_b_s[qp1q];
                        b_b_s[qp1q] := b_b_s[qq];
                        b_b_s[qq] := rt;
                        i0_xswap(x := Vf, ix0 := (5 * qp1q) + 1, iy0 := (5 * (qp1q + 1)) + 1);
                        i0_xswap_g(x := U, ix0 := (6 * qp1q) + 1, iy0 := (6 * (qp1q + 1)) + 1);
                        qp1q := qq;
                        qq := qq + 1;
                    ELSE 
                        exitg1 := 1;
                    END_IF;
                ELSE 
                    exitg1 := 1;
                END_IF;
            UNTIL NOT(exitg1 = 0)
            END_REPEAT;
            qq := 0;
            m := m - 1;
    END_CASE;
END_WHILE;
FOR m := 0 TO 4 DO 
    b_s[m] := b_b_s[m];
    FOR qq := 0 TO 4 DO 
        V[qq + (5 * m)] := Vf[(5 * m) + qq];
    END_FOR;
END_FOR;

END_FUNCTION_BLOCK

// ---- KinematicsForwAndInverseMatLab/xrot_c.TcPOU
FUNCTION_BLOCK xrot_c
VAR_INPUT
    ix0: DINT;
    iy0: DINT;
    c: LREAL;
    b_s: LREAL;
END_VAR
VAR_IN_OUT
    x: ARRAY [0..29] OF LREAL;
END_VAR
VAR_TEMP
    k: DINT;
    temp_tmp: DINT;
    temp_tmp_0: LREAL;
    temp_tmp_1: DINT;
    temp_tmp_2: LREAL;
END_VAR

FOR k := 0 TO 5 DO 
    temp_tmp := (iy0 + k) - 1;
    temp_tmp_0 := x[temp_tmp];
    temp_tmp_1 := (ix0 + k) - 1;
    temp_tmp_2 := x[temp_tmp_1];
    x[temp_tmp] := (temp_tmp_0 * c) - (temp_tmp_2 * b_s);
    x[temp_tmp_1] := (temp_tmp_2 * c) + (temp_tmp_0 * b_s);
END_FOR;

END_FUNCTION_BLOCK

// ---- KinematicsForwAndInverseMatLab/xrotg.TcPOU
FUNCTION_BLOCK xrotg
VAR_OUTPUT
    c: LREAL;
    b_s: LREAL;
END_VAR
VAR_IN_OUT
    a: LREAL;
    b: LREAL;
END_VAR
VAR_TEMP
    roe: LREAL;
    absa: LREAL;
    absb: LREAL;
    scale: LREAL;
    ads: LREAL;
    bds: LREAL;
END_VAR

roe := b;
absa := ABS(a);
absb := ABS(b);
IF absa > absb THEN 
    roe := a;
END_IF;
scale := absa + absb;
IF scale = 0.0 THEN 
    b_s := 0.0;
    c := 1.0;
    a := 0.0;
    b := 0.0;
ELSE 
    ads := absa / scale;
    bds := absb / scale;
    scale := SQRT((ads * ads) + (bds * bds)) * scale;
    IF roe < 0.0 THEN 
        scale :=  -scale;
    END_IF;
    c := a / scale;
    b_s := b / scale;
    IF absa > absb THEN 
        b := b_s;
    ELSIF c <> 0.0 THEN 
        b := 1.0 / c;
    ELSE 
        b := 1.0;
    END_IF;
    a := scale;
END_IF;

END_FUNCTION_BLOCK

// ---- KinematicsForwAndInverseMatLab/xrot.TcPOU
FUNCTION_BLOCK xrot
VAR_INPUT
    ix0: DINT;
    iy0: DINT;
    c: LREAL;
    b_s: LREAL;
END_VAR
VAR_IN_OUT
    x: ARRAY [0..24] OF LREAL;
END_VAR
VAR_TEMP
    k: DINT;
    temp_tmp: DINT;
    temp_tmp_0: LREAL;
    temp_tmp_1: DINT;
    temp_tmp_2: LREAL;
END_VAR

FOR k := 0 TO 4 DO 
    temp_tmp := (iy0 + k) - 1;
    temp_tmp_0 := x[temp_tmp];
    temp_tmp_1 := (ix0 + k) - 1;
    temp_tmp_2 := x[temp_tmp_1];
    x[temp_tmp] := (temp_tmp_0 * c) - (temp_tmp_2 * b_s);
    x[temp_tmp_1] := (temp_tmp_2 * c) + (temp_tmp_0 * b_s);
END_FOR;

END_FUNCTION_BLOCK

// ---- KinematicsForwAndInverseMatLab/xswap_g.TcPOU
FUNCTION_BLOCK xswap_g
VAR_INPUT
    ix0: DINT;
    iy0: DINT;
END_VAR
VAR_IN_OUT
    x: ARRAY [0..29] OF LREAL;
END_VAR
VAR_TEMP
    temp: LREAL;
    k: DINT;
    temp_tmp: DINT;
    tmp: DINT;
END_VAR

FOR k := 0 TO 5 DO 
    temp_tmp := (ix0 + k) - 1;
    temp := x[temp_tmp];
    tmp := (iy0 + k) - 1;
    x[temp_tmp] := x[tmp];
    x[tmp] := temp;
END_FOR;

END_FUNCTION_BLOCK

// ---- KinematicsForwAndInverseMatLab/xswap.TcPOU
FUNCTION_BLOCK xswap
VAR_INPUT
    ix0: DINT;
    iy0: DINT;
END_VAR
VAR_IN_OUT
    x: ARRAY [0..24] OF LREAL;
END_VAR
VAR_TEMP
    temp: LREAL;
    k: DINT;
    temp_tmp: DINT;
    tmp: DINT;
END_VAR

FOR k := 0 TO 4 DO 
    temp_tmp := (ix0 + k) - 1;
    temp := x[temp_tmp];
    tmp := (iy0 + k) - 1;
    x[temp_tmp] := x[tmp];
    x[tmp] := temp;
END_FOR;

END_FUNCTION_BLOCK

// ---- KinematicsForwAndInverseMatLab/xscal_fiz.TcPOU
FUNCTION_BLOCK xscal_fiz
VAR_INPUT
    a: LREAL;
    ix0: DINT;
END_VAR
VAR_IN_OUT
    x: ARRAY [0..24] OF LREAL;
END_VAR
VAR_TEMP
    k: DINT;
END_VAR

k := ix0;
WHILE k <= (ix0 + 4) DO
    x[k - 1] := x[k - 1] * a;
    k := k + 1;
END_WHILE;

END_FUNCTION_BLOCK

// ---- KinematicsForwAndInverseMatLab/xscal_fi.TcPOU
FUNCTION_BLOCK xscal_fi
VAR_INPUT
    a: LREAL;
    ix0: DINT;
END_VAR
VAR_IN_OUT
    x: ARRAY [0..29] OF LREAL;
END_VAR
VAR_TEMP
    k: DINT;
END_VAR

k := ix0;
WHILE k <= (ix0 + 5) DO
    x[k - 1] := x[k - 1] * a;
    k := k + 1;
END_WHILE;

END_FUNCTION_BLOCK

// ---- KinematicsForwAndInverseMatLab/xaxpy_dmy.TcPOU
FUNCTION_BLOCK xaxpy_dmy
VAR_INPUT
    b_n: DINT;
    a: LREAL;
    ix0: DINT;
    iy0: DINT;
END_VAR
VAR_IN_OUT
    y: ARRAY [0..24] OF LREAL;
END_VAR
VAR_TEMP
    ix: DINT;
    iy: DINT;
    k: DINT;
END_VAR

IF (b_n >= 1) AND (a <> 0.0) THEN 
    ix := ix0 - 1;
    iy := iy0 - 1;
    k := 0;
    WHILE k <= (b_n - 1) DO
        y[iy] := (a * y[ix]) + y[iy];
        ix := ix + 1;
        iy := iy + 1;
        k := k + 1;
    END_WHILE;
END_IF;

END_FUNCTION_BLOCK

// ---- KinematicsForwAndInverseMatLab/xaxpy.TcPOU
FUNCTION_BLOCK xaxpy
VAR_INPUT
    b_n: DINT;
    a: LREAL;
    ix0: DINT;
    iy0: DINT;
END_VAR
VAR_IN_OUT
    y: ARRAY [0..29] OF LREAL;
END_VAR
VAR_TEMP
    ix: DINT;
    iy: DINT;
    k: DINT;
END_VAR

IF (b_n >= 1) AND (a <> 0.0) THEN 
    ix := ix0 - 1;
    iy := iy0 - 1;
    k := 0;
    WHILE k <= (b_n - 1) DO
        y[iy] := (a * y[ix]) + y[iy];
        ix := ix + 1;
        iy := iy + 1;
        k := k + 1;
    END_WHILE;
END_IF;

END_FUNCTION_BLOCK

// ---- KinematicsForwAndInverseMatLab/xaxpy_d.TcPOU
FUNCTION_BLOCK xaxpy_d
VAR_INPUT
    b_n: DINT;
    a: LREAL;
    x: ARRAY [0..29] OF LREAL;
    ix0: DINT;
    iy0: DINT;
END_VAR
VAR_IN_OUT
    y: ARRAY [0..5] OF LREAL;
END_VAR
VAR_TEMP
    ix: DINT;
    iy: DINT;
    k: DINT;
END_VAR

IF (b_n >= 1) AND (a <> 0.0) THEN 
    ix := ix0 - 1;
    iy := iy0 - 1;
    k := 0;
    WHILE k <= (b_n - 1) DO
        y[iy] := (a * x[ix]) + y[iy];
        ix := ix + 1;
        iy := iy + 1;
        k := k + 1;
    END_WHILE;
END_IF;

END_FUNCTION_BLOCK

// ---- KinematicsForwAndInverseMatLab/xaxpy_dm.TcPOU
FUNCTION_BLOCK xaxpy_dm
VAR_INPUT
    b_n: DINT;
    a: LREAL;
    x: ARRAY [0..5] OF LREAL;
    ix0: DINT;
    iy0: DINT;
END_VAR
VAR_IN_OUT
    y: ARRAY [0..29] OF LREAL;
END_VAR
VAR_TEMP
    ix: DINT;
    iy: DINT;
    k: DINT;
END_VAR

IF (b_n >= 1) AND (a <> 0.0) THEN 
    ix := ix0 - 1;
    iy := iy0 - 1;
    k := 0;
    WHILE k <= (b_n - 1) DO
        y[iy] := (a * x[ix]) + y[iy];
        ix := ix + 1;
        iy := iy + 1;
        k := k + 1;
    END_WHILE;
END_IF;

END_FUNCTION_BLOCK

// ---- KinematicsForwAndInverseMatLab/xscal_f.TcPOU
FUNCTION_BLOCK xscal_f
VAR_INPUT
    b_n: DINT;
    a: LREAL;
    ix0: DINT;
END_VAR
VAR_IN_OUT
    x: ARRAY [0..4] OF LREAL;
END_VAR
VAR_TEMP
    b: DINT;
    k: DINT;
END_VAR

b := (ix0 + b_n) - 1;
k := ix0;
WHILE k <= b DO
    x[k - 1] := x[k - 1] * a;
    k := k + 1;
END_WHILE;

END_FUNCTION_BLOCK

// ---- KinematicsForwAndInverseMatLab/xscal.TcPOU
FUNCTION_BLOCK xscal
VAR_INPUT
    b_n: DINT;
    a: LREAL;
    ix0: DINT;
END_VAR
VAR_IN_OUT
    x: ARRAY [0..29] OF LREAL;
END_VAR
VAR_TEMP
    b: DINT;
    k: DINT;
END_VAR

b := (ix0 + b_n) - 1;
k := ix0;
WHILE k <= b DO
    x[k - 1] := x[k - 1] * a;
    k := k + 1;
END_WHILE;

END_FUNCTION_BLOCK

// ---- KinematicsForwAndInverseMatLab/xnrm2.TcPOU
FUNCTION xnrm2 : LREAL
VAR_INPUT
    b_n: DINT;
    x: ARRAY [0..29] OF LREAL;
    ix0: DINT;
END_VAR
VAR
    scale: LREAL;
    kend: DINT;
    absxk: LREAL;
    t: LREAL;
    k: DINT;
END_VAR

xnrm2 := 0.0;
IF b_n >= 1 THEN 
    IF b_n = 1 THEN 
        xnrm2 := ABS(x[ix0 - 1]);
    ELSE 
        scale := 3.3121686421112381E-170;
        kend := (ix0 + b_n) - 1;
        k := ix0;
        WHILE k <= kend DO
            absxk := ABS(x[k - 1]);
            IF absxk > scale THEN 
                t := scale / absxk;
                xnrm2 := ((xnrm2 * t) * t) + 1.0;
                scale := absxk;
            ELSE 
                t := absxk / scale;
                xnrm2 := (t * t) + xnrm2;
            END_IF;
            k := k + 1;
        END_WHILE;
        xnrm2 := scale * SQRT(xnrm2);
    END_IF;
END_IF;

END_FUNCTION

// ---- KinematicsForwAndInverseMatLab/xdotc.TcPOU
FUNCTION xdotc : LREAL
VAR_INPUT
    b_n: DINT;
    x: ARRAY [0..29] OF LREAL;
    ix0: DINT;
    y: ARRAY [0..29] OF LREAL;
    iy0: DINT;
END_VAR
VAR
    ix: DINT;
    iy: DINT;
    k: DINT;
END_VAR

xdotc := 0.0;
IF b_n >= 1 THEN 
    ix := ix0;
    iy := iy0;
    k := 0;
    WHILE k <= (b_n - 1) DO
        xdotc := (x[ix - 1] * y[iy - 1]) + xdotc;
        ix := ix + 1;
        iy := iy + 1;
        k := k + 1;
    END_WHILE;
END_IF;

END_FUNCTION

// ---- KinematicsForwAndInverseMatLab/xnrm2_l.TcPOU
FUNCTION xnrm2_l : LREAL
VAR_INPUT
    b_n: DINT;
    x: ARRAY [0..4] OF LREAL;
    ix0: DINT;
END_VAR
VAR
    scale: LREAL;
    kend: DINT;
    absxk: LREAL;
    t: LREAL;
    k: DINT;
END_VAR

xnrm2_l := 0.0;
IF b_n >= 1 THEN 
    IF b_n = 1 THEN 
        xnrm2_l := ABS(x[ix0 - 1]);
    ELSE 
        scale := 3.3121686421112381E-170;
        kend := (ix0 + b_n) - 1;
        k := ix0;
        WHILE k <= kend DO
            absxk := ABS(x[k - 1]);
            IF absxk > scale THEN 
                t := scale / absxk;
                xnrm2_l := ((xnrm2_l * t) * t) + 1.0;
                scale := absxk;
            ELSE 
                t := absxk / scale;
                xnrm2_l := (t * t) + xnrm2_l;
            END_IF;
            k := k + 1;
        END_WHILE;
        xnrm2_l := scale * SQRT(xnrm2_l);
    END_IF;
END_IF;

END_FUNCTION

// ---- KinematicsForwAndInverseMatLab/xdotc_i.TcPOU
FUNCTION xdotc_i : LREAL
VAR_INPUT
    b_n: DINT;
    x: ARRAY [0..24] OF LREAL;
    ix0: DINT;
    y: ARRAY [0..24] OF LREAL;
    iy0: DINT;
END_VAR
VAR
    ix: DINT;
    iy: DINT;
    k: DINT;
END_VAR

xdotc_i := 0.0;
IF b_n >= 1 THEN 
    ix := ix0;
    iy := iy0;
    k := 0;
    WHILE k <= (b_n - 1) DO
        xdotc_i := (x[ix - 1] * y[iy - 1]) + xdotc_i;
        ix := ix + 1;
        iy := iy + 1;
        k := k + 1;
    END_WHILE;
END_IF;

END_FUNCTION

// ---- KinematicsForwAndInverseMatLab/eps.TcPOU
FUNCTION eps : LREAL
VAR_INPUT
    x: LREAL;
END_VAR
VAR
    absx: LREAL;
    exponent: DINT;
    ln2x: LREAL;
    e: DINT;
    temp15: LREAL;
END_VAR

absx := ABS(x);
IF absx < 2.2250738585072014E-307 THEN 
    eps := 2.2250738585072014E-307;
ELSE 
    temp15 := LN(absx);
    ln2x := rt_floord(u := temp15 / 0.69314718055994529);
    exponent := TRUNC(ln2x) - 1;
    e :=  -TRUNC(ln2x);
    IF ( -TRUNC(ln2x)) < -1022 THEN 
        absx := absx * 1.90109156629516E-211;
        e := 700 - TRUNC(ln2x);
        IF (700 - TRUNC(ln2x)) < -1022 THEN 
            absx := absx * 1.90109156629516E-211;
            e := 1400 - TRUNC(ln2x);
        END_IF;
    ELSIF ( -TRUNC(ln2x)) > 1023 THEN 
        absx := absx * 5.2601359015483735E+210;
        e := ( -TRUNC(ln2x)) - 700;
        IF (( -TRUNC(ln2x)) - 700) > 1023 THEN 
            absx := absx * 5.2601359015483735E+210;
            e := ( -TRUNC(ln2x)) - 1400;
        END_IF;
    END_IF;
    absx := absx * EXPT(2.0, DINT_TO_LREAL(e));
    IF absx < 0.5 THEN 
        exponent := TRUNC(ln2x) - 2;
    ELSIF absx >= 1.0 THEN 
        exponent := TRUNC(ln2x);
    END_IF;
    eps := rt_ldexp_U1d_U2s32_Yd_s_pw(u0 := 1.0, u1 := exponent - 52);
END_IF;

END_FUNCTION

// ---- KinematicsForwAndInverseMatLab/rt_floord.TcPOU
FUNCTION rt_floord : LREAL
VAR_INPUT
    u: LREAL;
END_VAR

rt_floord := DINT_TO_LREAL(TRUNC(u));
IF u = rt_floord THEN 
    rt_floord := u;
ELSIF u < 0.0 THEN 
    rt_floord := rt_floord - 1.0;
END_IF;

END_FUNCTION

// ---- KinematicsForwAndInverseMatLab/rt_ldexp_U1d_U2s32_Yd_s_pw.TcPOU
FUNCTION rt_ldexp_U1d_U2s32_Yd_s_pw : LREAL
VAR_INPUT
    u0: LREAL;
    u1: DINT;
END_VAR

IF (u0 = 0.0) OR (u1 = 0) THEN 
    rt_ldexp_U1d_U2s32_Yd_s_pw := u0;
ELSE 
    rt_ldexp_U1d_U2s32_Yd_s_pw := u0 * EXPT(2.0, DINT_TO_LREAL(u1));
END_IF;

END_FUNCTION

// ---- KinematicsForwAndInverseMatLab/pinv_i.TcPOU
FUNCTION_BLOCK pinv_i
VAR_INPUT
    A: ARRAY [0..35] OF LREAL;
END_VAR
VAR_OUTPUT
    X: ARRAY [0..35] OF LREAL;
END_VAR
VAR
    i0_svd_e: svd_e;
END_VAR
VAR_TEMP
    V: ARRAY [0..35] OF LREAL;
    b_r: DINT;
    vcol: DINT;
    U: ARRAY [0..35] OF LREAL;
    b_s: ARRAY [0..5] OF LREAL;
    tol: LREAL;
    j: DINT;
    ar: DINT;
    ia: DINT;
    b: DINT;
    ib: DINT;
    b_ic: DINT;
    exitg1: DINT;
END_VAR

b_r := -1;
FOR vcol := 0 TO 35 DO 
    X[vcol] := 0.0;
END_FOR;
i0_svd_e(A := A);
U := i0_svd_e.U;
b_s := i0_svd_e.b_s;
V := i0_svd_e.V;
tol := 6.0 * eps(x := b_s[0]);
vcol := 0;
REPEAT 
    exitg1 := 0;
    IF vcol < 6 THEN 
        IF b_s[vcol] <= tol THEN 
            exitg1 := 1;
        ELSE 
            b_r := b_r + 1;
            vcol := vcol + 1;
        END_IF;
    ELSE 
        exitg1 := 1;
    END_IF;
UNTIL NOT(exitg1 = 0)
END_REPEAT;
IF (b_r + 1) > 0 THEN 
    vcol := 0;
    j := 0;
    WHILE j <= b_r DO
        tol := 1.0 / b_s[j];
        ar := vcol;
        WHILE (ar + 1) <= (vcol + 6) DO
            V[ar] := tol * V[ar];
            ar := ar + 1;
        END_WHILE;
        vcol := vcol + 6;
        j := j + 1;
    END_WHILE;
    vcol := 0;
    FOR j := 0 TO 31 BY 6 DO 
        ar := j;
        WHILE (ar + 1) <= (j + 6) DO
            X[ar] := 0.0;
            ar := ar + 1;
        END_WHILE;
    END_FOR;
    FOR j := 0 TO 31 BY 6 DO 
        ar := -1;
        vcol := vcol + 1;
        b := (6 * b_r) + vcol;
        ib := vcol;
        WHILE ib <= b DO
            ia := ar;
            b_ic := j;
            WHILE (b_ic + 1) <= (j + 6) DO
                ia := ia + 1;
                X[b_ic] := (U[ib - 1] * V[ia]) + X[b_ic];
                b_ic := b_ic + 1;
            END_WHILE;
            ar := ar + 6;
            ib := ib + 6;
        END_WHILE;
    END_FOR;
END_IF;

END_FUNCTION_BLOCK

// ---- KinematicsForwAndInverseMatLab/svd_e.TcPOU
FUNCTION_BLOCK svd_e
VAR_INPUT
    A: ARRAY [0..35] OF LREAL;
END_VAR
VAR_OUTPUT
    U: ARRAY [0..35] OF LREAL;
    b_s: ARRAY [0..5] OF LREAL;
    V: ARRAY [0..35] OF LREAL;
END_VAR
VAR
    i0_xrot_c5: xrot_c5;
    i0_xrotg: xrotg;
    i0_xswap_gs: xswap_gs;
    i0_xscal_fiz1t4: xscal_fiz1t4;
    i0_xaxpy_dmyz: xaxpy_dmyz;
    i0_xaxpy_dmyzr: xaxpy_dmyzr;
    i0_xaxpy_dmyzr5: xaxpy_dmyzr5;
    i0_xscal_fiz1t: xscal_fiz1t;
    i0_xscal_fiz1: xscal_fiz1;
END_VAR
VAR_TEMP
    b_A: ARRAY [0..35] OF LREAL;
    b_b_s: ARRAY [0..5] OF LREAL;
    e: ARRAY [0..5] OF LREAL;
    work: ARRAY [0..5] OF LREAL;
    Vf: ARRAY [0..35] OF LREAL;
    qq: DINT;
    apply_transform: BOOL;
    nrm: LREAL;
    qjj: DINT;
    qp1jj: DINT;
    m: DINT;
    qp1q: DINT;
    rt: LREAL;
    ztest: LREAL;
    smm1: LREAL;
    emm1: LREAL;
    sqds: LREAL;
    shift: LREAL;
    k_ii: DINT;
    exitg1: DINT;
    temp16: LREAL;
    temp17: LREAL;
    temp18: LREAL;
    temp19: LREAL;
    temp20: LREAL;
    temp21: LREAL;
    temp22: LREAL;
    temp23: LREAL;
    temp24: LREAL;
    temp25: LREAL;
    temp26: LREAL;
    temp27: LREAL;
    temp28: LREAL;
    temp29: LREAL;
END_VAR

